ABB RobotStudio station: Braižymas_Paletavimas_V_Januška.rspag

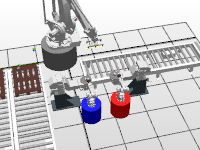
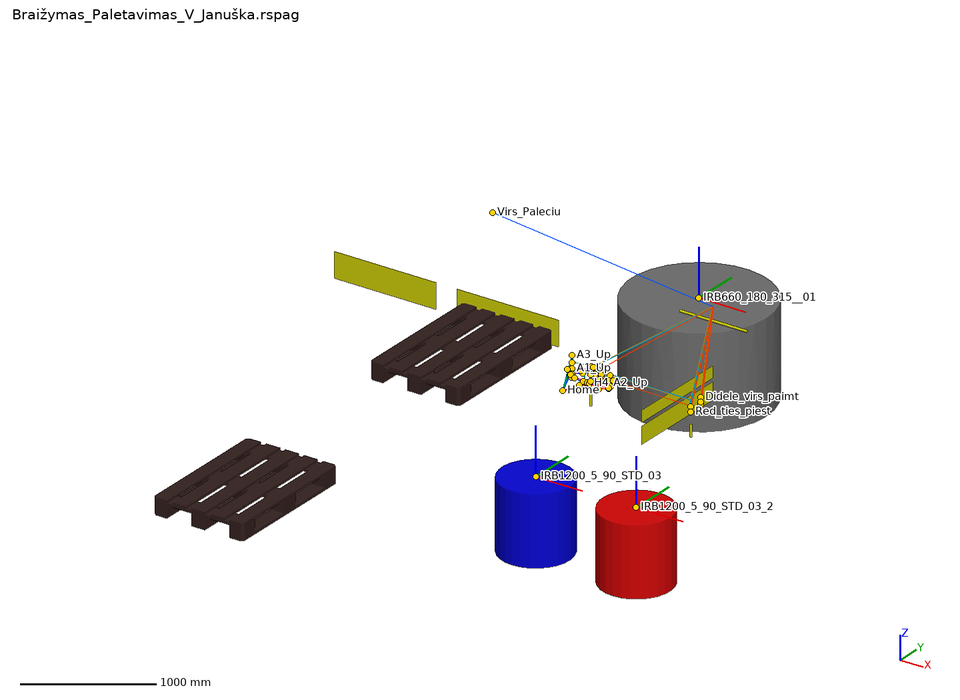
[picture v1: parts stored in the station drawn from their meshes, with robot base, taught points and paths (robot models come from the ABB library and are not in the file)]
--- station ---
Station Braižymas_Paletavimas_V_Januška (saved by RobotStudio 21.4.9700.0)
Controller Paint_Red, task T_ROB1: task frame (RAPID world) sits at (1200, -2800, 600) mm, rotated rx 0 ry 0 rz 90 deg in the station
Controller Paint_Blue, task T_ROB1: task frame (RAPID world) sits at (300, -2800, 600) mm, rotated rx 0 ry 0 rz 90 deg in the station
Controller Paletavimas, task T_ROB1: task frame (RAPID world) sits at (-200, 0, 0) mm, rotated rx 0 ry 0 rz 180 deg in the station
Controller Paletavimas
  mechanical unit ROB_1: IRB660_180_315__01, 6 joints, base frame (0, 0, 800) mm
Controller Paint_Blue
  mechanical unit ROB_1: IRB1200_5_90_STD_03, 6 joints, base frame (0, 0, 0) mm
Controller Paint_Red
  mechanical unit ROB_1: IRB1200_5_90_STD_03_2, 6 joints, base frame (0, 0, 0) mm
Layout (positions relative to the parent item):
  - IRB660_180_315__01 [mechanism] at (-200, 0, 800) mm, rotated rx 0 ry 0 rz 180 deg; joint values [2.2494, 0.0329, 0.7758, 0.6816] (rad or m)
      links: Base, Link1, Link2, Link3, LinkD1, LinkD2, LinkS1, LinkS2, Link4, LinkS3, Link6, LinkS4, LinkS5
  - Pakyla [part] at (-200, 0, 0) mm, size 1200 x 1200 x 800 mm
  - Conveyor_EUR_SC [smart component] at (-1000, -4700, 0) mm, rotated rx 0 ry 0 rz 90 deg
      signals: DI DI_New_Box, DO DO_Box_In_Place, DI DI_Delete_Pallet
      connections:
        Conveyor_EUR_SC.DI_New_Box -> PalletSource.Execute
        PalletSource.Executed -> PalletQueue.Enqueue
        PalletPlaneSensor.SensorOut -> PalletQueue.Dequeue
        PalletPlaneSensor.SensorOut -> Conveyor_EUR_SC.DO_Box_In_Place
        PalletPlaneSensor.SensorOut -> LogicGate.InputA
        LogicGate.Output -> PalletSource.Execute
        Conveyor_EUR_SC.DI_Delete_Pallet -> Sink.Execute
        PalletSource.Copy => PalletQueue.Back
        PalletPlaneSensor.SensedPart => Sink.Object
    - 950_4000_h2 [part, from Equipment\Conveyor 950 4000 h2.rslib]
    - PalletSource [smart component, from Components\Source.rslib] at (90, 55, 415) mm
        properties: Source=Euro Pallet; Copy=(none); Parent=(none); Position=[0.09 0.055 0.415]; Orientation=[0 0 0]; Transient=false; PhysicsBehavior=0
    - PalletQueue [smart component, from Components\Queue.rslib]
        properties: Back=(none); Front=(none); Queue={971251d9-3e66-4420-9243-4213e4a19f12}; NumberOfObjects=1
    - PalletPlaneSensor [smart component, from Components\PlaneSensor.rslib]
        properties: Origin=[4.05 0 0.436]; Axis1=[0 0.91 0]; Axis2=[0 0 0.22]; SensedPart=Body 1
      - _sensorPart_ [part], size 0 x 910 x 220 mm
    - LogicGate [smart component, from Components\LogicGate.rslib]
        properties: Operator=NOT; Delay=0
    - LinearMover [smart component, from Components\LinearMover.rslib]
        properties: Object=PalletQueue; Direction=[0 0.001 0]; Speed=1.2; Reference=Global; ReferenceObject=(none)
    - Euro Pallet [graphiccomponentgroup] at (90, 55, 415) mm
      - Body 1 [part], size 1200 x 800 x 144 mm
    - Sink [smart component, from Components\Sink.rslib]
        properties: Object=Body 1
    - Euro Pallet_2 [graphiccomponentgroup] at (2854.8, 55, 415) mm
      - Body 1 [part], size 1200 x 800 x 144 mm
  - Conveyor_EUR_Tall_SC [smart component] at (-2100, -4700, 0) mm, rotated rx 0 ry 0 rz 90 deg
      signals: DI DI_New_Box, DO DO_Box_In_Place, DI DI_Delete_Pallet
      connections:
        Conveyor_EUR_Tall_SC.DI_New_Box -> PalletSource.Execute
        PalletSource.Executed -> PalletQueue.Enqueue
        PalletPlaneSensor.SensorOut -> PalletQueue.Dequeue
        PalletPlaneSensor.SensorOut -> Conveyor_EUR_Tall_SC.DO_Box_In_Place
        PalletPlaneSensor.SensorOut -> LogicGate.InputA
        LogicGate.Output -> PalletSource.Execute
        Conveyor_EUR_Tall_SC.DI_Delete_Pallet -> Sink.Execute
        PalletSource.Copy => PalletQueue.Back
        PalletPlaneSensor.SensedPart => Sink.Object
    - 950_4000_h2 [part, from Equipment\Conveyor 950 4000 h2.rslib]
    - PalletSource [smart component, from Components\Source.rslib] at (90, 55, 415) mm
        properties: Source=Euro Pallet; Copy=Euro Pallet_6; Parent=(none); Position=[0.09 0.055 0.415]; Orientation=[0 0 0]; Transient=false; PhysicsBehavior=0
    - PalletQueue [smart component, from Components\Queue.rslib]
        properties: Back=Euro Pallet_6; Front=(none); Queue=; NumberOfObjects=0
    - PalletPlaneSensor [smart component, from Components\PlaneSensor.rslib]
        properties: Origin=[4.05 0 0.436]; Axis1=[0 0.91 0]; Axis2=[0 0 0.22]; SensedPart=Body 1
      - _sensorPart_ [part], size 0 x 910 x 220 mm
    - LogicGate [smart component, from Components\LogicGate.rslib]
        properties: Operator=NOT; Delay=0
    - LinearMover [smart component, from Components\LinearMover.rslib]
        properties: Object=PalletQueue; Direction=[0 0.001 0]; Speed=1.2; Reference=Global; ReferenceObject=(none)
    - Euro Pallet [graphiccomponentgroup, from Equipment\Euro Pallet.rslib] at (90, 55, 415) mm
      - Body 1 [part, from Equipment\Euro Pallet.rslib]
    - Sink [smart component, from Components\Sink.rslib]
        properties: Object=Body 1
    - Euro Pallet_6 [graphiccomponentgroup, from Equipment\Euro Pallet.rslib] at (2854.8, 55, 415) mm
      - Body 1 [part, from Equipment\Euro Pallet.rslib]
  - Pakyla_2 [part] at (300, -2800, 0) mm, rotated rx 0 ry 0 rz -90 deg, size 600 x 599 x 600 mm
  - Pakyla_3 [part] at (3000, -1800, 0) mm, rotated rx 0 ry 0 rz -90 deg, size 600 x 599 x 600 mm
  - Griebtuvas_2 [smart component] at (-790.8, -1192.17, 822.02) mm
      signals: DI DI_Attach, DI DI_Enque_Tall, DI DI_Enque_Small, DI DI_Delete_Small, DI DI_Delete_Tall
      connections:
        Griebtuvas_2.DI_Attach -> PoseMover_2.Execute
        Griebtuvas_2.DI_Attach -> Attacher.Execute
        Griebtuvas_2.DI_Attach -> LogicGate.InputA
        LogicGate.Output -> Detacher.Execute
        Griebtuvas_2.DI_Enque_Tall -> Delete_Tall_Queue.Enqueue
        Griebtuvas_2.DI_Enque_Small -> Delete_Small_Queue.Enqueue
        Griebtuvas_2.DI_Delete_Small -> Delete_Small_Queue.DeleteAll
        Griebtuvas_2.DI_Delete_Tall -> Delete_Tall_Queue.DeleteAll
        LineSensor.SensedPart => Detacher.Child
        LineSensor.SensedPart => Attacher.Child
        LineSensor.SensedPart => Delete_Small_Queue.Back
        LineSensor.SensedPart => Delete_Tall_Queue.Back
    - Attacher [smart component, from Components\Attacher.rslib] at (1573.68, -26.65, 864.9) mm, rotated rx 180 ry 0 rz 89.83 deg
        properties: Parent=Griebtuvas_2; Flange=0; Child=(none); Mount=false; Offset=[0 0 0]; Orientation=[0 0 0]
    - Detacher [smart component, from Components\Detacher.rslib] at (1573.68, -26.65, 864.9) mm, rotated rx 180 ry 0 rz 89.83 deg
        properties: Child=(none); KeepPosition=true
    - LineSensor [smart component, from Components\LineSensor.rslib] at (1573.68, -26.65, 864.9) mm, rotated rx 180 ry 0 rz 89.83 deg
        properties: Start=[-6.04715178049997E-07 0.300000227208211 0.311447110706865]; End=[-3.13979206786885E-07 -0.300000333635623 0.311447110706865]; Radius=0.01; SensedPart=(none); SensedPoint=[0 0 0]
      - _sensorPart_ [part], size 20 x 600 x 20 mm
    - VacuumTool [mechanism] at (1573.68, -26.65, 864.9) mm, rotated rx 180 ry 0 rz 89.83 deg
        TCP tVacuum at (0, 0, 200) mm
        links: VacuumTool
    - LogicGate [smart component, from Components\LogicGate.rslib]
        properties: Operator=NOT; Delay=0
    - Delete_Small_Queue [smart component, from Components\Queue.rslib]
        properties: Back=(none); Front=(none); Queue=; NumberOfObjects=0
    - Delete_Tall_Queue [smart component, from Components\Queue.rslib]
        properties: Back=(none); Front=(none); Queue=; NumberOfObjects=0
  - Pozicionierius_Red [smart component] at (1200, -2100, 0) mm
      signals: DI DI_Attach, DO DO_Attached, DI DI_TurnR, DI DI_TurnL, DO DO_Complete, DI DI_Home, DO DO_Free
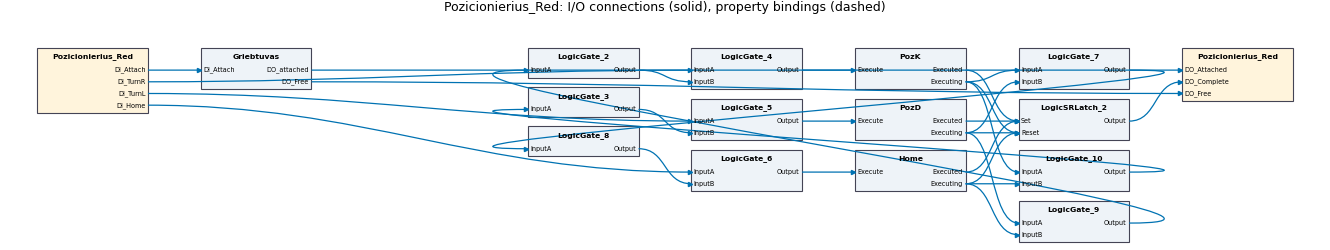
      connections:
        Pozicionierius_Red.DI_Attach -> Griebtuvas.DI_Attach
        Griebtuvas.DO_attached -> Pozicionierius_Red.DO_Attached
        LogicGate_4.Output -> PozK.Execute
        LogicGate_5.Output -> PozD.Execute
        LogicGate_6.Output -> Home.Execute
        Pozicionierius_Red.DI_TurnR -> LogicGate_4.InputA
        Pozicionierius_Red.DI_TurnL -> LogicGate_5.InputA
        Pozicionierius_Red.DI_Home -> LogicGate_6.InputA
        LogicSRLatch_2.Output -> Pozicionierius_Red.DO_Complete
        PozK.Executed -> LogicSRLatch_2.Set
        PozD.Executed -> LogicSRLatch_2.Set
        Home.Executed -> LogicSRLatch_2.Set
        PozK.Executing -> LogicGate_7.InputA
        PozK.Executing -> LogicGate_10.InputA
        PozD.Executing -> LogicGate_7.InputB
        PozD.Executing -> LogicGate_9.InputA
        Home.Executing -> LogicGate_9.InputB
        Home.Executing -> LogicGate_10.InputB
        LogicGate_9.Output -> LogicGate_2.InputA
        LogicGate_10.Output -> LogicGate_3.InputA
        LogicGate_7.Output -> LogicGate_8.InputA
        LogicGate_2.Output -> LogicGate_4.InputB
        LogicGate_3.Output -> LogicGate_5.InputB
        LogicGate_8.Output -> LogicGate_6.InputB
        Home.Executing -> LogicSRLatch_2.Reset
        PozD.Executing -> LogicSRLatch_2.Reset
        PozK.Executing -> LogicSRLatch_2.Reset
        Griebtuvas.DO_Free -> Pozicionierius_Red.DO_Free
    - Griebtuvas [smart component]
        signals: DI DI_Attach, DO DO_attached, DO DO_Free
        connections:
          Griebtuvas.DI_Attach -> Attacher.Execute
          Griebtuvas.DI_Attach -> LogicGate.InputA
          LogicGate.Output -> Detacher.Execute
          Attacher.Executed -> LogicSRLatch.Set
          Detacher.Executed -> LogicSRLatch.Reset
          LogicSRLatch.Output -> Griebtuvas.DO_attached
          LineSensor.SensorOut -> LogicGate_2.InputA
          LogicGate_2.Output -> Griebtuvas.DO_Free
          LineSensor.SensedPart => Attacher.Child
          LineSensor.SensedPart => Detacher.Child
      - Attacher [smart component, from Components\Attacher.rslib]
          properties: Parent=IRBP_A250_D1000_M2009_REV1_01; Flange=0; Child=(none); Mount=false; Offset=[0 0 0]; Orientation=[0 0 0]
      - Detacher [smart component, from Components\Detacher.rslib]
          properties: Child=(none); KeepPosition=true
      - LogicGate [smart component, from Components\LogicGate.rslib]
          properties: Operator=NOT; Delay=0
      - LogicSRLatch [smart component, from Components\LogicSRLatch.rslib]
      - LineSensor [smart component, from Components\LineSensor.rslib]
          properties: Start=[0 0 0.9]; End=[0 0 1]; Radius=0.01; SensedPart=(none); SensedPoint=[0 0 0]
        - _sensorPart_ [part], size 20 x 20 x 100 mm
      - LogicGate_2 [smart component, from Components\LogicGate.rslib]
          properties: Operator=NOT; Delay=0
    - IRBP_A250_D1000_M2009_REV1_01 [mechanism] at (0, 0, 0) mm; joint values [0, 1.5708] (rad or m)
        links: Base, Link1, Link2
    - PozD [smart component, from Components\PoseMover.rslib]
        properties: Mechanism=IRBP_A250_D1000_M2009_REV1_01; Pose=2; Duration=0.5
    - PozK [smart component, from Components\PoseMover.rslib]
        properties: Mechanism=IRBP_A250_D1000_M2009_REV1_01; Pose=3; Duration=0.5
    - Home [smart component, from Components\PoseMover.rslib]
        properties: Mechanism=IRBP_A250_D1000_M2009_REV1_01; Pose=1; Duration=0.5
    - LogicGate_2 [smart component, from Components\LogicGate.rslib]
        properties: Operator=NOT; Delay=0
    - LogicGate_3 [smart component, from Components\LogicGate.rslib]
        properties: Operator=NOT; Delay=0
    - LogicGate_4 [smart component, from Components\LogicGate.rslib]
        properties: Operator=AND; Delay=0
    - LogicGate_5 [smart component, from Components\LogicGate.rslib]
        properties: Operator=AND; Delay=0
    - LogicGate_6 [smart component, from Components\LogicGate.rslib]
        properties: Operator=AND; Delay=0
    - LogicGate_7 [smart component, from Components\LogicGate.rslib]
        properties: Operator=OR; Delay=0
    - LogicGate_8 [smart component, from Components\LogicGate.rslib]
        properties: Operator=NOT; Delay=0
    - LogicGate_9 [smart component, from Components\LogicGate.rslib]
        properties: Operator=OR; Delay=0
    - LogicGate_10 [smart component, from Components\LogicGate.rslib]
        properties: Operator=OR; Delay=0
    - LogicSRLatch_2 [smart component, from Components\LogicSRLatch.rslib]
  - Pozicionierius_Blue [smart component] at (300, -2100, 0) mm, rotated rx 0 ry 0 rz 180 deg
      signals: DI DI_Attach, DO DO_Attached, DI DI_TurnR, DI DI_TurnL, DO DO_Complete, DI DI_Home, DO DO_Free
      connections:
        Pozicionierius_Blue.DI_Attach -> Griebtuvas.DI_Attach
        Griebtuvas.DO_attached -> Pozicionierius_Blue.DO_Attached
        LogicGate_4.Output -> PozK.Execute
        LogicGate_5.Output -> PozD.Execute
        LogicGate_6.Output -> Home.Execute
        Pozicionierius_Blue.DI_TurnR -> LogicGate_4.InputA
        Pozicionierius_Blue.DI_TurnL -> LogicGate_5.InputA
        Pozicionierius_Blue.DI_Home -> LogicGate_6.InputA
        LogicSRLatch_2.Output -> Pozicionierius_Blue.DO_Complete
        PozK.Executed -> LogicSRLatch_2.Set
        PozD.Executed -> LogicSRLatch_2.Set
        Home.Executed -> LogicSRLatch_2.Set
        PozK.Executing -> LogicGate_7.InputA
        PozK.Executing -> LogicGate_10.InputA
        PozD.Executing -> LogicGate_7.InputB
        PozD.Executing -> LogicGate_9.InputA
        Home.Executing -> LogicGate_9.InputB
        Home.Executing -> LogicGate_10.InputB
        LogicGate_9.Output -> LogicGate_2.InputA
        LogicGate_10.Output -> LogicGate_3.InputA
        LogicGate_7.Output -> LogicGate_8.InputA
        LogicGate_2.Output -> LogicGate_4.InputB
        LogicGate_3.Output -> LogicGate_5.InputB
        LogicGate_8.Output -> LogicGate_6.InputB
        Home.Executing -> LogicSRLatch_2.Reset
        PozD.Executing -> LogicSRLatch_2.Reset
        PozK.Executing -> LogicSRLatch_2.Reset
        Griebtuvas.DO_Free -> Pozicionierius_Blue.DO_Free
    - Griebtuvas [smart component]
        signals: DI DI_Attach, DO DO_attached, DO DO_Free
        connections:
          Griebtuvas.DI_Attach -> Attacher.Execute
          Griebtuvas.DI_Attach -> LogicGate.InputA
          LogicGate.Output -> Detacher.Execute
          Attacher.Executed -> LogicSRLatch.Set
          Detacher.Executed -> LogicSRLatch.Reset
          LogicSRLatch.Output -> Griebtuvas.DO_attached
          LineSensor.SensorOut -> LogicGate_3.InputA
          LogicGate_3.Output -> Griebtuvas.DO_Free
          LineSensor.SensedPart => Attacher.Child
          LineSensor.SensedPart => Detacher.Child
          LineSensor.SensedPart => Detacher.Child
          LineSensor.SensedPart => Attacher.Child
      - Attacher [smart component, from Components\Attacher.rslib]
          properties: Parent=IRBP_A250_D1000_M2009_REV1_01; Flange=0; Child=(none); Mount=false; Offset=[0 0 0]; Orientation=[0 0 0]
      - Detacher [smart component, from Components\Detacher.rslib]
          properties: Child=(none); KeepPosition=true
      - LogicGate [smart component, from Components\LogicGate.rslib]
          properties: Operator=NOT; Delay=0
      - LogicSRLatch [smart component, from Components\LogicSRLatch.rslib]
      - LineSensor [smart component, from Components\LineSensor.rslib]
          properties: Start=[0 0 0.9]; End=[0 0 1]; Radius=0.01; SensedPart=(none); SensedPoint=[0 0 0]
        - _sensorPart_ [part], size 20 x 20 x 100 mm
      - LogicGate_3 [smart component, from Components\LogicGate.rslib]
          properties: Operator=NOT; Delay=0
    - IRBP_A250_D1000_M2009_REV1_01 [mechanism] at (0, 0, 0) mm; joint values [0, 1.5708] (rad or m)
        links: Base, Link1, Link2
    - PozD [smart component, from Components\PoseMover.rslib]
        properties: Mechanism=IRBP_A250_D1000_M2009_REV1_01; Pose=2; Duration=0.5
    - PozK [smart component, from Components\PoseMover.rslib]
        properties: Mechanism=IRBP_A250_D1000_M2009_REV1_01; Pose=3; Duration=0.5
    - Home [smart component, from Components\PoseMover.rslib]
        properties: Mechanism=IRBP_A250_D1000_M2009_REV1_01; Pose=1; Duration=0.5
    - LogicGate_2 [smart component, from Components\LogicGate.rslib]
        properties: Operator=NOT; Delay=0
    - LogicGate_3 [smart component, from Components\LogicGate.rslib]
        properties: Operator=NOT; Delay=0
    - LogicGate_4 [smart component, from Components\LogicGate.rslib]
        properties: Operator=AND; Delay=0
    - LogicGate_5 [smart component, from Components\LogicGate.rslib]
        properties: Operator=AND; Delay=0
    - LogicGate_6 [smart component, from Components\LogicGate.rslib]
        properties: Operator=AND; Delay=0
    - LogicGate_7 [smart component, from Components\LogicGate.rslib]
        properties: Operator=OR; Delay=0
    - LogicGate_8 [smart component, from Components\LogicGate.rslib]
        properties: Operator=NOT; Delay=0
    - LogicGate_9 [smart component, from Components\LogicGate.rslib]
        properties: Operator=OR; Delay=0
    - LogicGate_10 [smart component, from Components\LogicGate.rslib]
        properties: Operator=OR; Delay=0
    - LogicSRLatch_2 [smart component, from Components\LogicSRLatch.rslib]
  - IRB1200_5_90_STD_03 [mechanism, from Robots\IRB1200_5_90_STD_03.rslib] at (300, -2800, 600) mm, rotated rx 0 ry 0 rz 90 deg; joint values [-0.0192, -0.8245, 0.9777, -0.1248, -0.1544, 0.1234] (rad or m)
  - IRB1200_5_90_STD_03_2 [mechanism, from Robots\IRB1200_5_90_STD_03.rslib] at (1200, -2800, 600) mm, rotated rx 0 ry 0 rz 90 deg; joint values [-0.0192, -0.8245, 0.9777, -0.1248, -0.1544, 0.1234] (rad or m)
  - Conveyor_RND_SC [smart component] at (4500, -750, 0) mm, rotated rx 0 ry 0 rz 180 deg
      signals: DI DI_New_Box, DO DO_Box_InPlace, DO DO_TallBox_InPlace, DO DO_Only_High_Sensor
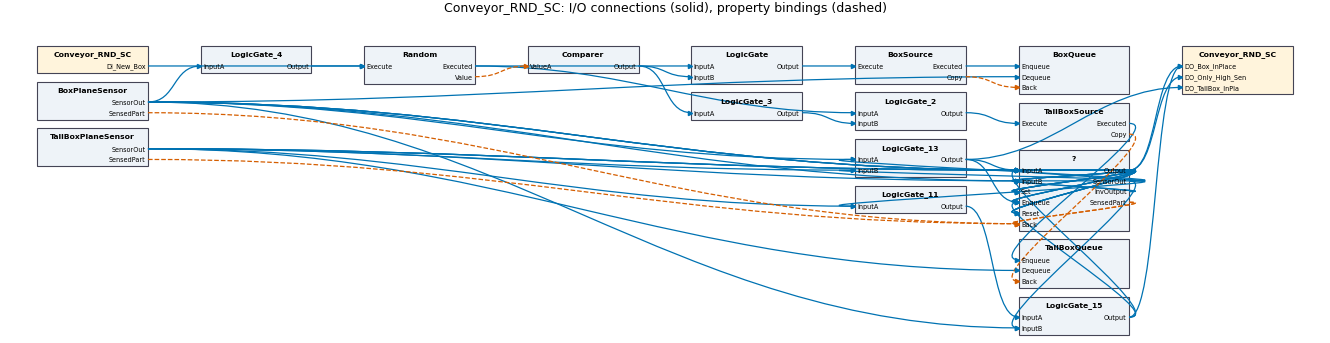
      connections:
        Conveyor_RND_SC.DI_New_Box -> Random.Execute
        Random.Executed -> LogicGate.InputA
        Random.Executed -> LogicGate_2.InputA
        Comparer.Output -> LogicGate_3.InputA
        LogicGate_3.Output -> LogicGate_2.InputB
        Comparer.Output -> LogicGate.InputB
        LogicGate.Output -> BoxSource.Execute
        LogicGate_2.Output -> TallBoxSource.Execute
        BoxSource.Executed -> BoxQueue.Enqueue
        LogicGate_4.Output -> Random.Execute
        BoxPlaneSensor.SensorOut -> LogicGate_4.InputA
        BoxPlaneSensor.SensorOut -> BoxQueue.Dequeue
        TallBoxSource.Executed -> TallBoxQueue.Enqueue
        TallBoxPlaneSensor.SensorOut -> TallBoxQueue.Dequeue
        TallBoxPlaneSensor.SensorOut -> ?.InputA
        BoxPlaneSensor.SensorOut -> ?.InputA
        ?.Output -> ?.InputB
        TallBoxPlaneSensor.SensorOut -> ?.InputA
        BoxPlaneSensor.SensorOut -> ?.InputB
        ?.Output -> ?.InputA
        ?.Output -> ?.Set
        ?.Output -> Conveyor_RND_SC.DO_Box_InPlace
        ?.Output -> Delete_Small_Queue.Enqueue
        ?.Output -> ?.Set
        ?.Output -> ?.InputA
        ?.Output -> ?.Reset
        ?.Output -> ?.InputA
        ?.Output -> ?.Reset
        ?.SensorOut -> LogicGate_13.InputA
        ?.SensorOut -> LogicGate_13.InputB
        ?.SensorOut -> LogicGate_11.InputA
        LogicGate_11.Output -> LogicGate_15.InputA
        ?.SensorOut -> LogicGate_15.InputB
        LogicGate_13.Output -> LogicGate_16.InputA
        LogicGate_16.Output -> LogicSRLatch_4.Set
        LogicGate_15.Output -> LogicGate_14.InputA
        LogicGate_14.Output -> LogicSRLatch_5.Set
        LogicSRLatch_5.InvOutput -> LogicGate_16.InputB
        LogicSRLatch_4.InvOutput -> LogicGate_14.InputB
        ?.SensorOut -> LogicGate_18.InputA
        ?.SensorOut -> LogicGate_18.InputB
        LogicGate_18.Output -> LogicGate_17.InputA
        LogicGate_17.Output -> LogicSRLatch_4.Reset
        TallBoxPlaneSensor.SensorOut -> LogicGate_18.InputB
        TallBoxPlaneSensor.SensorOut -> LogicGate_13.InputB
        TallBoxPlaneSensor.SensorOut -> LogicGate_11.InputA
        BoxPlaneSensor.SensorOut -> LogicGate_18.InputA
        BoxPlaneSensor.SensorOut -> LogicGate_13.InputA
        BoxPlaneSensor.SensorOut -> LogicGate_15.InputB
        LogicSRLatch_5.Output -> LogicGate_19.InputB
        LogicGate_19.Output -> Delete_Small_Queue.Enqueue
        LogicGate_20.Output -> Delete_Tall_Queue.Enqueue
        LogicSRLatch_4.Output -> LogicGate_20.InputB
        LogicGate_23.Output -> LogicGate_21.InputB
        BoxPlaneSensor.SensorOut -> LogicGate_23.InputA
        TallBoxPlaneSensor.SensorOut -> LogicGate_21.InputA
        LogicGate_21.Output -> LogicGate_19.InputA
        LogicGate_21.Output -> LogicGate_20.InputA
        LogicGate_21.Output -> Conveyor_RND_SC.DO_Only_High_Sensor
        LogicGate_17.Output -> LogicSRLatch_5.Reset
        LogicGate_13.Output -> Conveyor_RND_SC.DO_TallBox_InPlace
        LogicGate_15.Output -> Conveyor_RND_SC.DO_Box_InPlace
        LogicGate_15.Output -> Delete_Small_Queue.Enqueue
        LogicGate_13.Output -> Delete_Tall_Queue.Enqueue
        Random.Value => Comparer.ValueA
        BoxSource.Copy => BoxQueue.Back
        TallBoxSource.Copy => TallBoxQueue.Back
        DeleteSensor.SensedPart => Delete_Small_Queue.Back
        DeleteSensor.SensedPart => Delete_Tall_Queue.Back
        BoxPlaneSensor.SensedPart => Delete_Small_Queue.Back
        TallBoxPlaneSensor.SensedPart => Delete_Tall_Queue.Back
    - 950_4000 [part, from Equipment\Conveyor 950 4000 h2.rslib]
    - Box [part] at (60, 300, 415) mm, size 500 x 300 x 200 mm
    - BoxPlaneSensor [smart component, from Components\PlaneSensor.rslib]
        properties: Origin=[4.05 0 0.45]; Axis1=[0 0.91 0]; Axis2=[0 0 0.15]; SensedPart=(none)
      - _sensorPart_ [part], size 0 x 910 x 150 mm
    - BoxQueue [smart component, from Components\Queue.rslib] at (0, -3000, 0) mm
        properties: Back=(none); Front=(none); Queue={fa6990f4-df59-49ae-9a32-9599613f68ec};{e767133d-be7e-453b-8722-821a6b4558c0};{6ce431a7-dd26-4a38-b4fa-eec74b1977cf};{3ae16747-654e-4202-adcd-dee3cf7f9746};{658dea4e-2eb4-4657-ae88-8a3f4d155435};{5f69d4f6-3337-4fea-9838-df10eb0f07de};{5aecbc6f-cfd0-44df-ba1d-f4507ba342ea};{9e44f664-69de-4a1f-8895-3168aa3968ee};{5f2001e6-6928-42db-81b0-89c8c28d3b67};{af1fb1b9-f86a-429e-8c15-d7efb4d2c7e7};{8385d1b0-8c34-4fb9-9887-15fbe6147db4};{4006f633-1bd4-4d72-a937-3620dfa0b835};{8730c694-ac09-41e2-b981-cff9bcc11746};{a723061a-c6e3-4254-9954-9e38f42a9860};{04c40ebc-cfd0-4884-a185-3f6b111fdaa2};{a878a6d6-609e-42c1-80c8-878f67ab97da};{14d7b2c0-999e-4cbf-889d-0a124069ec19};{0becc2c0-5e92-4cfa-b639-036a75e5a4e4};{cca5aef1-b22d-4971-98ab-11323a0a7094};{e02a7358-ec92-4485-b2c0-c2038150d912};{6839aee3-4009-4411-9cbe-94a25d9f948c};{9f3facf0-270c-4be3-a67a-821ea0c5aa08};{faba08c9-aeb2-4eb9-b9c7-e387a6e9cbfb};{bc03e252-87de-4255-9640-78523ef2143d};{aa76d2e2-ad85-4407-8279-2d879163961a};{be818020-9745-4898-a081-c1837189eb10};{37e33ad3-8b58-4812-a8ee-bee1f17e24b7};{41a75c38-fc95-4d9b-aee3-f79fb853da63};{f3c5d293-df41-45c9-8c8c-c5c112b7c860};{0c1f799b-0fa7-450f-a03e-204d5134bc88};{4de367fb-fa00-4147-a461-8cdc53a5ab36};{fb4f46fb-3cc9-46d0-93b3-3697bff4c5b0};{1981477c-fa3d-405d-81ed-5c11cf4004f1};{4a3acb3a-f0fe-49f4-bb5a-d33d1ebb5bdb};{ee543a3a-f0a7-4b8a-ba73-df8df06667eb};{37d46d93-7b88-48c0-95e4-0c0aea62eed6};{e38b9446-edb0-4063-af88-28e337124caa};{43dc83e6-1610-4f95-90e3-0b23558226fe};{ea22c4f6-820c-436e-a9cf-17bec50e4e45};{7837ae08-a857-4e45-b104-d71f85b8db14};{a15a4319-5ddc-4b41-a9f1-f3fc310fac6a};{fcbb5e9a-b5e8-401e-bfdc-b057d8770794};{ce142922-48a3-4377-89ec-985408ba8153};{9c2054a3-2d81-4b78-8319-3879110db110};{4184086f-4b9b-435c-872e-61dbf8e8b281};{2e9da51f-8d60-4fa4-b223-03c706fc42b4};{f081e902-d69f-44bb-8e7e-e42cb8ba28a7};{0c45a0ca-c831-4e04-b0c0-ea9f274c986f};{68cd1851-b56a-466d-8aa0-fcc04310c142};{8d21e733-4511-40ca-a380-e002fb2e741f};{1fdcc6e5-ab2a-4a16-b63c-6443d12e6cd0};{928b3c83-786f-4b1b-b774-b6e363eb8edd};{c5d4ec7b-f50e-4586-9c9a-3cfc5369afde};{176768ad-9249-4043-a0f4-b263c87cbf02};{a41bf4c8-ca06-40df-8d99-855080af08cc};{1f7c0284-63bf-491f-a88a-99226beab572};{93b63075-c389-479b-b9ba-db424c8f1608};{46184e33-de41-46df-bfa5-1fa5c4186c93};{ff1b25a2-d9f1-4991-8a41-ba89a23b8150};{72555af7-e6df-461e-9b88-b16b7a0d81b3};{b15f7b76-8d34-4692-97fc-69f520f0f3c0};{93a6a054-f8ca-4001-a03b-5df487de4b8b};{72ed48d2-5bfa-4ecc-a1ec-2e7778b8ef55};{9cda9d10-0121-4b20-9212-f063ab80550a};{33ea0952-9bf3-4e06-b34c-2e0ac0a36824};{e1a11204-25f8-485f-a139-3d4a140b070a};{3c953577-cf61-4183-9ff0-bca456af431b};{30fbd990-83ea-4ba2-9465-f98aa0538540};{dfe653b7-7d94-4ddd-b2ef-7199ad70201c};{82d208d8-4dee-4044-8917-702fcaee31aa};{aa19c751-7ff3-4b4e-bfb3-31ee09fcbfd8};{cfec794f-833e-41bb-b0d0-1a3d28b30ff6};{6a23a3bd-1c81-490c-bc0d-d6dcbd6c3643};{8a1ebaad-f4c7-4178-a576-8aee444642b5};{ba785cc5-e159-446c-93f0-7483d17038e5};{828e2240-582c-4548-b989-1a7bc8d860a3};{4a59a418-7f0b-41e9-93ce-595c45a59b07};{f4dbaa99-1c72-4e73-8856-0fc6635ef423};{6087b47d-53c7-4741-b2a3-0c083e370b15};{2e30bba9-a6bf-4b01-9fc0-a1f4cbfc7dfc};{19071a2c-5ad0-42a1-9bd2-bb839ae9b4d4};{b0002f64-93e0-428c-b2e5-2d4d9f7da933};{a347c7fd-09d1-4374-ab85-2149f88733a9};{b0d38dbd-07a6-4783-b2e8-5f2c5d6b0201};{2266d51d-b3d0-4d52-bbb5-de615e632cc2};{75460951-9708-49ff-8c70-7d7735d8d5c2};{295ff81f-2104-47a7-8bd3-4eaad3dc957a};{0a807d55-7f1b-46ac-9050-abab5979a08e};{896dd1f3-c715-442d-b525-9d9e6cb6e06f};{4fa8727e-168a-49f4-b20a-f869ddebea6d};{9c068a76-23d8-4921-84fc-952de2f64cfe};{4b6f13b1-b58b-4cfc-9d2f-06395fabde15};{01d6ab25-4f5e-4e9f-bdfc-4dfebc0f0cf6};{0ab7461e-d2ad-4383-836c-68a8b79c7dca};{06b8ba49-82c0-4634-8553-9497b791d1b9};{f3c0ef50-404a-451a-a529-2526a8561f87};{0ffca263-bbd3-4c7e-912c-55349d3e2daa};{252a513a-a084-4872-865a-129838c2f94f};{466e5942-a908-47e1-8cd1-136cfa812536};{1b8b29c7-edcf-413e-9f81-164808a08126};{5c9bba4a-b90c-47ae-95ca-d31383bcbc95};{a37f6f99-c3a3-4e91-9e81-52d69c79e6c0};{eaa8d07c-22f4-4512-a4ed-d3e2fd25e17b};{cd5a02a4-7d6b-4818-9494-1cca1ee745c5};{c0bf9634-2c95-4f7a-b6ff-e31064599eb0};{8cba37ce-13ba-401a-b10d-a55bd7da9434};{350e1ddc-e127-4834-bdb0-6da9a5ae8f39};{12ff0c17-9d1a-4539-a0c4-b273c13be77a};{36d11481-6af8-4316-a391-be7944f9a913};{9e99407b-b875-4dbb-ac3e-7ed2c2198c50};{18fd7586-1f58-49bb-aa86-4785e5672a8a};{4590a0b8-4fa4-4fd5-96ec-6588471226b3};{0910f9d0-3289-4e14-ada6-3d436962069f};{6e596c34-5dbf-4a37-9b92-6d9d57f91504};{2fc5be82-8ebc-4497-b7a2-a92180d8126c};{e572f00d-1eb5-4a34-a751-0ba51d1a1975};{68969745-703d-4f84-abfd-8cca6df6441f};{bd9b3794-10fd-4df4-8bef-e9c82c14e8cf};{f3ae70ba-db38-470f-8edb-540b6fe1d8be};{2a3c6a5a-be7f-42bd-82e9-81bfd16108a1};{25c3ed99-c921-4982-a94c-124f118646ae}; NumberOfObjects=1
    - BoxSource [smart component, from Components\Source.rslib] at (0, -3000, 0) mm
        properties: Source=Box; Copy=(none); Parent=(none); Position=[0.06 0.325 0.415]; Orientation=[0 0 0]; Transient=false; PhysicsBehavior=0
    - LinearMover [smart component, from Components\LinearMover.rslib] at (0, -3000, 0) mm
        properties: Object=BoxQueue; Direction=[-0.001 0 0]; Speed=1.2; Reference=Global; ReferenceObject=(none)
    - Random [smart component, from Components\Random.rslib] at (3800, -500, 0) mm, rotated rx 0 ry 0 rz 180 deg
        properties: Value=0.429773476640588; Min=0; Max=1
    - Comparer [smart component, from Components\Comparer.rslib] at (3800, -500, 0) mm, rotated rx 0 ry 0 rz 180 deg
        properties: ValueA=0.429773476640588; Operator=>=; ValueB=0.5
    - TallBoxSource [smart component, from Components\Source.rslib] at (0, -3000, 0) mm
        properties: Source=Box_tall; Copy=(none); Parent=(none); Position=[0.06 0.325 0.415]; Orientation=[0 0 0]; Transient=false; PhysicsBehavior=0
    - LogicGate [smart component, from Components\LogicGate.rslib] at (3800, -500, 0) mm, rotated rx 0 ry 0 rz 180 deg
        properties: Operator=AND; Delay=0
    - LogicGate_2 [smart component, from Components\LogicGate.rslib] at (3800, -500, 0) mm, rotated rx 0 ry 0 rz 180 deg
        properties: Operator=AND; Delay=0
    - LogicGate_3 [smart component, from Components\LogicGate.rslib] at (3800, -500, 0) mm, rotated rx 0 ry 0 rz 180 deg
        properties: Operator=NOT; Delay=0
    - LogicGate_4 [smart component, from Components\LogicGate.rslib] at (3800, -500, 0) mm, rotated rx 0 ry 0 rz 180 deg
        properties: Operator=NOT; Delay=0
    - TallBoxPlaneSensor [smart component, from Components\PlaneSensor.rslib]
        properties: Origin=[4.05 0 0.63]; Axis1=[0 0.91 0]; Axis2=[0 0 0.1]; SensedPart=(none)
      - _sensorPart_ [part], size 0 x 910 x 100 mm
    - Box_tall [part] at (60, 300, 415) mm, size 500 x 300 x 250 mm
    - TallBoxQueue [smart component, from Components\Queue.rslib]
        properties: Back=(none); Front=(none); Queue=; NumberOfObjects=0
    - LinearMover_2 [smart component, from Components\LinearMover.rslib]
        properties: Object=TallBoxQueue; Direction=[-0.001 0 0]; Speed=1.2; Reference=Global; ReferenceObject=(none)
    - LogicGate_10 [smart component, from Components\LogicGate.rslib]
        properties: Operator=AND; Delay=0
    - LogicGate_11 [smart component, from Components\LogicGate.rslib]
        properties: Operator=NOT; Delay=0
    - LogicGate_12 [smart component, from Components\LogicGate.rslib]
        properties: Operator=AND; Delay=0
    - LogicGate_13 [smart component, from Components\LogicGate.rslib]
        properties: Operator=AND; Delay=0
    - LogicGate_15 [smart component, from Components\LogicGate.rslib]
        properties: Operator=AND; Delay=0
  - TraceTCP [smart component, from Components\TraceTCP.rslib]
      properties: Robot=IRB1200_5_90_STD_03
  - TraceTCP_2 [smart component, from Components\TraceTCP.rslib]
      properties: Robot=IRB1200_5_90_STD_03_2
  - Pen_Blue [mechanism, from Training Objects\Pen.rslib] at (302.36, -2594.82, 1275.93) mm, rotated rx 0 ry 90 rz 90 deg
  - Pen_Red [mechanism, from Training Objects\Pen.rslib] at (1202.36, -2594.82, 1275.93) mm, rotated rx 0 ry 90 rz 90 deg
Attachment: VacuumTool is attached to IRB660_180_315__01 / Link6
Attachment: Griebtuvas_2 is attached to IRB660_180_315__01 / Link6
Attachment: TallBoxSource is attached to BoxSource
Attachment: Pen_Blue is attached to IRB1200_5_90_STD_03 / Link6
Attachment: Pen_Red is attached to IRB1200_5_90_STD_03_2 / Link6
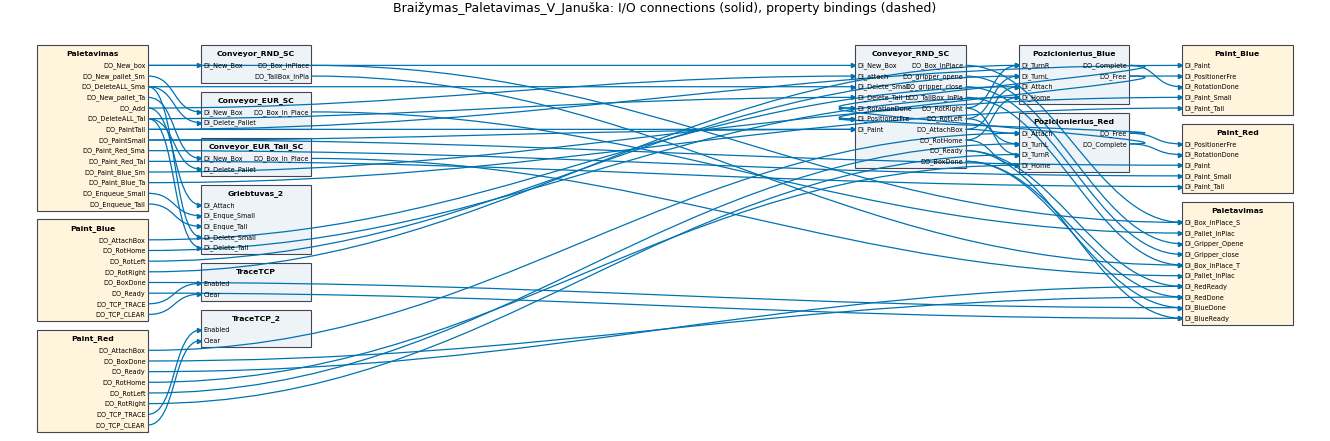
Station logic (signal -> signal, property => property):
  Paletavimas.DO_New_box -> Conveyor_RND_SC.DI_New_Box
  Paletavimas.DO_New_pallet_Small -> Conveyor_EUR_SC.DI_New_Box
  Conveyor_RND_SC.DO_Box_InPlace -> Paletavimas.DI_Box_InPlace_Small
  Conveyor_EUR_SC.DO_Box_In_Place -> Paletavimas.DI_Pallet_InPlace_Small
  Griebtuvas_SC.DO_gripper_opened -> Paletavimas.DI_Gripper_Opened
  Griebtuvas_SC.DO_gripper_closed -> Paletavimas.DI_Gripper_closed
  Paletavimas.DO_DeleteALL_Small -> Conveyor_EUR_SC.DI_Delete_Pallet
  Paletavimas.DO_New_pallet_Tall -> Conveyor_EUR_Tall_SC.DI_New_Box
  Conveyor_RND_SC.DO_TallBox_InPlace -> Paletavimas.DI_Box_InPlace_Tall
  Conveyor_EUR_Tall_SC.DO_Box_In_Place -> Paletavimas.DI_Pallet_InPlace_Tall
  Paletavimas.DO_Add -> Griebtuvas_SC.DI_attach
  Paletavimas.DO_DeleteALL_Tall -> Conveyor_EUR_Tall_SC.DI_Delete_Pallet
  Paletavimas.DO_DeleteALL_Small -> Conveyor_RND_SC.DI_Delete_Small_boxes
  Paletavimas.DO_DeleteALL_Tall -> Conveyor_RND_SC.DI_Delete_Tall_boxes
  Piesimas_Blue.DO_RotRight -> Pozicionierius_Blue.DI_TurnR
  Piesimas_Blue.DO_RotLeft -> Pozicionierius_Blue.DI_TurnL
  Piesimas_Red.DO_AttachBox -> Pozicionierius_Red.DI_Attach
  Piesimas_Blue.DO_AttachBox -> Pozicionierius_Blue.DI_Attach
  Paletavimas.DO_Add -> Griebtuvas_2.DI_Attach
  Piesimas_Blue.DO_RotHome -> Pozicionierius_Blue.DI_Home
  Pozicionierius_Blue.DO_Complete -> Piesimas_Blue.DI_RotationDone
  Pozicionierius_Blue.DO_Free -> Piesimas_Blue.DI_PositionerFree
  Piesimas_Red.DO_RotLeft -> Pozicionierius_Red.DI_TurnL
  Piesimas_Red.DO_RotRight -> Pozicionierius_Red.DI_TurnR
  Piesimas_Red.DO_RotHome -> Pozicionierius_Red.DI_Home
  Pozicionierius_Red.DO_Free -> Piesimas_Red.DI_PositionerFree
  Pozicionierius_Red.DO_Complete -> Piesimas_Red.DI_RotationDone
  Piesimas_Red.DO_Ready -> Paletavimas.DI_RedReady
  Piesimas_Red.DO_BoxDone -> Paletavimas.DI_RedDone
  Piesimas_Blue.DO_BoxDone -> Paletavimas.DI_BlueDone
  Piesimas_Blue.DO_Ready -> Paletavimas.DI_BlueReady
  Paletavimas.DO_PaintTall -> Piesimas_Blue.DI_Paint
  Paletavimas.DO_PaintSmall -> Piesimas_Red.DI_Paint
  Paint_Blue.DO_AttachBox -> Pozicionierius_Blue.DI_Attach
  Paint_Blue.DO_RotHome -> Pozicionierius_Blue.DI_Home
  Paint_Blue.DO_RotLeft -> Pozicionierius_Blue.DI_TurnL
  Paint_Blue.DO_RotRight -> Pozicionierius_Blue.DI_TurnR
  Paint_Blue.DO_BoxDone -> Paletavimas.DI_BlueDone
  Paletavimas.DO_PaintTall -> Paint_Blue.DI_Paint
  Pozicionierius_Blue.DO_Free -> Paint_Blue.DI_PositionerFree
  Pozicionierius_Blue.DO_Complete -> Paint_Blue.DI_RotationDone
  Paint_Red.DO_AttachBox -> Pozicionierius_Red.DI_Attach
  Paint_Red.DO_BoxDone -> Paletavimas.DI_RedDone
  Paint_Red.DO_Ready -> Paletavimas.DI_RedReady
  Paint_Red.DO_RotHome -> Pozicionierius_Red.DI_Home
  Paint_Red.DO_RotLeft -> Pozicionierius_Red.DI_TurnL
  Paint_Red.DO_RotRight -> Pozicionierius_Red.DI_TurnR
  Pozicionierius_Red.DO_Free -> Paint_Red.DI_PositionerFree
  Pozicionierius_Red.DO_Complete -> Paint_Red.DI_RotationDone
  Paletavimas.DO_PaintSmall -> Paint_Red.DI_Paint
  Conveyor_RND_SC.DO_Box_InPlace -> Paletavimas.DI_Box_InPlace_Small
  Conveyor_RND_SC.DO_TallBox_InPlace -> Paletavimas.DI_Box_InPlace_Tall
  Paletavimas.DO_New_box -> Conveyor_RND_SC.DI_New_Box
  Paint_Blue.DO_Ready -> Paletavimas.DI_BlueReady
  Paint_Blue.DO_TCP_TRACE -> TraceTCP.Enabled
  Paint_Blue.DO_TCP_CLEAR -> TraceTCP.Clear
  Paint_Red.DO_TCP_TRACE -> TraceTCP_2.Enabled
  Paint_Red.DO_TCP_CLEAR -> TraceTCP_2.Clear
  Paletavimas.DO_Paint_Red_Small -> Paint_Red.DI_Paint_Small
  Paletavimas.DO_Paint_Red_Tall -> Paint_Red.DI_Paint_Tall
  Paletavimas.DO_Paint_Blue_Small -> Paint_Blue.DI_Paint_Small
  Paletavimas.DO_Paint_Blue_Tall -> Paint_Blue.DI_Paint_Tall
  Paletavimas.DO_Enqueue_Small -> Griebtuvas_2.DI_Enque_Small
  Paletavimas.DO_Enqueue_Tall -> Griebtuvas_2.DI_Enque_Tall
  Paletavimas.DO_DeleteALL_Small -> Griebtuvas_2.DI_Delete_Small
  Paletavimas.DO_DeleteALL_Tall -> Griebtuvas_2.DI_Delete_Tall
Targets, tools, work objects and paths stored in the station and not in the controller backup, written as RAPID:
! task T_ROB1
MODULE Module1
  CONST robtarget Didele_ties_piest:=[[-500.000094663,2099.999976261,1150.000241875],[0,-0.706073245,0.708138808,0],[-1,0,0,0],[9E+09,9E+09,9E+09,9E+09,9E+09,9E+09]];
  CONST robtarget Didele_virs_piest:=[[-500.00009482,2100.000045238,1205.091525026],[0,-0.706073245,0.708138808,0],[-1,0,0,0],[9E+09,9E+09,9E+09,9E+09,9E+09,9E+09]];
  CONST robtarget Maza_ties_piest:=[[-1400.000277317,2100.000253447,1100.000411858],[0,-0.706073243,0.708138811,0],[-1,0,0,0],[9E+09,9E+09,9E+09,9E+09,9E+09,9E+09]];
  CONST robtarget Maza_virs_piest:=[[-1400.000277317,2100.00034861,1144.065558591],[0,-0.706073227,0.708138826,0],[-1,0,0,0],[9E+09,9E+09,9E+09,9E+09,9E+09,9E+09]];
  CONST robtarget Didele_ties_conveyor:=[[2504.292,960.385,809],[0,0,1,0],[-2,0,0,0],[9E+09,9E+09,9E+09,9E+09,9E+09,9E+09]];
  CONST robtarget Maza_pries_piesima:=[[-200.095627935,1365.111929006,1486.920311485],[0,-0.706073231,0.708138822,0],[-1,0,0,0],[9E+09,9E+09,9E+09,9E+09,9E+09,9E+09]];
  CONST robtarget Didele_pries_piesima:=[[-876.40010473,1225.00022946,1665.000321221],[0,-0.706073245,0.708138808,0],[-1,0,0,0],[9E+09,9E+09,9E+09,9E+09,9E+09,9E+09]];
  CONST robtarget Maza_ties_conveyor:=[[1443.841,905.155,755.519],[0,0,1,0],[-2,0,0,0],[9E+09,9E+09,9E+09,9E+09,9E+09,9E+09]];
  CONST robtarget Didele_1:=[[2505.32,794.624,809],[0,-0.707106781,0.707106781,0],[-2,0,-1,0],[9E+09,9E+09,9E+09,9E+09,9E+09,9E+09]];
  CONST robtarget Maza_1:=[[1405.32,794.624,759],[0,-0.707106781,0.707106781,0],[0,0,0,0],[9E+09,9E+09,9E+09,9E+09,9E+09,9E+09]];
  PROC Deze_Tall_iki_konvejerio()
    MoveL Home,v1000,z100,tVacuum\WObj:=wobj0;
    MoveL Didele_pries_piesima,v1000,z100,tVacuum\WObj:=wobj0;
    MoveL Didele_ties_piest,v1000,z100,tVacuum\WObj:=wobj0;
    MoveL Didele_virs_piest,v1000,z100,tVacuum\WObj:=wobj0;
    MoveJ Didele_ties_conveyor,v1000,z100,tVacuum\WObj:=wobj0;
  ENDPROC
  PROC Deze_Small_iki_konvejerio()
    MoveL Home,v1000,z100,tVacuum\WObj:=wobj0;
    MoveL Maza_pries_piesima,v1000,z100,tVacuum\WObj:=wobj0;
    MoveL Maza_ties_piest,v1000,z100,tVacuum\WObj:=wobj0;
    MoveL Maza_virs_piest,v1000,z100,tVacuum\WObj:=wobj0;
    MoveL Maza_ties_conveyor,v1000,z100,tVacuum\WObj:=wobj0;
    MoveL Maza_ties_conveyor,v1000,z100,tVacuum\WObj:=wobj0;
  ENDPROC
  PROC Deze_Small_iki_padeklo()
    MoveJ Home,v1000,z100,tVacuum\WObj:=wobj0;
    MoveJ Maza_virs_paimt,v1000,z100,tVacuum\WObj:=wobj0;
    MoveL Maza_ties_paimt,v1000,z100,tVacuum\WObj:=wobj0;
    MoveL Maza_virs_paimt,v1000,z100,tVacuum\WObj:=wobj0;
    MoveL Home,v1000,z100,tVacuum\WObj:=wobj0;
    MoveJ Maza_pries_piesima,v1000,z100,tVacuum\WObj:=wobj0;
    MoveJ Maza_virs_piest,v1000,z100,tVacuum\WObj:=wobj0;
    MoveL Maza_ties_piest,v1000,z100,tVacuum\WObj:=wobj0;
    MoveL Maza_ties_piest,v1000,z100,tVacuum\WObj:=wobj0;
    MoveJ Maza_pries_piesima,v1000,z100,tVacuum\WObj:=wobj0;
    MoveJ Home,v1000,z100,tVacuum\WObj:=wobj0;
  ENDPROC
  PROC Deze_Tall_iki_padeklo()
    MoveL Home,v1000,z100,tVacuum\WObj:=wobj0;
    MoveL Didele_virs_paimt,v1000,z100,tVacuum\WObj:=wobj0;
    MoveL Didele_ties_paimt,v1000,z100,tVacuum\WObj:=wobj0;
    MoveL Didele_virs_paimt,v1000,z100,tVacuum\WObj:=wobj0;
    MoveL Home,v1000,z100,tVacuum\WObj:=wobj0;
    MoveJ Didele_pries_piesima,v1000,z100,tVacuum\WObj:=wobj0;
    MoveL Didele_virs_piest,v1000,z100,tVacuum\WObj:=wobj0;
    MoveL Didele_ties_piest,v1000,z100,tVacuum\WObj:=wobj0;
    MoveL Didele_virs_piest,v1000,z100,tVacuum\WObj:=wobj0;
    MoveJ Didele_pries_piesima,v1000,z100,tVacuum\WObj:=wobj0;
    MoveJ Home,v1000,z100,tVacuum\WObj:=wobj0;
  ENDPROC
  PROC Dezes_Pattern()
    MoveL Didele_1,v1000,z100,tVacuum\WObj:=wobj0;
    MoveL Maza_1,v1000,z100,tVacuum\WObj:=wobj0;
  ENDPROC
  PROC Virs()
    MoveL Virs_Paleciu,v1000,z100,tVacuum\WObj:=wobj0;
  ENDPROC
ENDMODULE


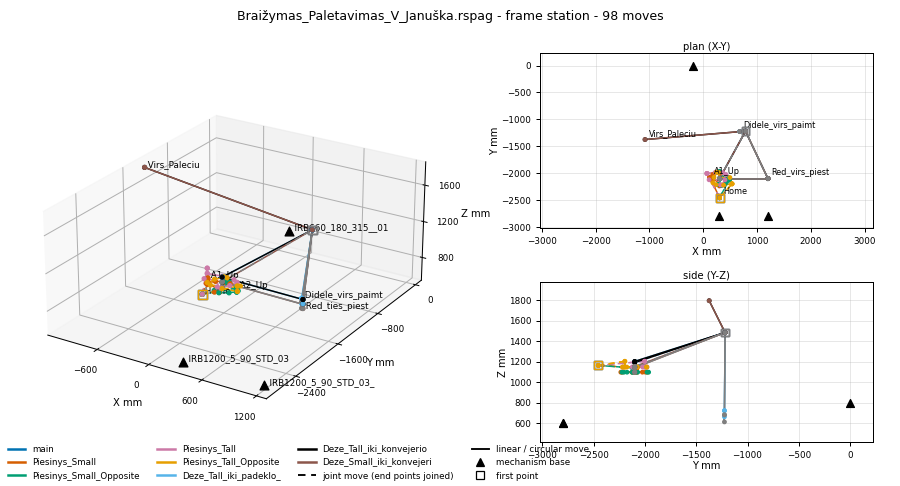
[picture p0: tool path of Braižymas_Paletavimas_V_Januška.rspag in frame station, 98 of 108 moves have a stored position in this frame; points joined in program order, loops and branches not executed]
--- Backups/Paint_Blue/RAPID/TASK1/PROGMOD/CalibData.mod ---
MODULE CalibData
    TASK PERS wobjdata Small_Dezes_Wobj:=[FALSE,TRUE,"",[[700,-800,-200],[0.707107,0,0,0.707107]],[[1050,150,700],[6.12323E-17,0,0,1]]];
    TASK PERS wobjdata Small_Dezes_Wobj_Op:=[FALSE,TRUE,"",[[0.137,-2.682,-3.962],[1,0,0,0]],[[849.863,-247.318,503.962],[0.707106781,0,0,0.707106781]]];
    TASK PERS wobjdata Tall_Dezes_Wobj:=[FALSE,TRUE,"",[[550,250,550],[0.707106781,0,0,-0.707106781]],[[0,0,0],[1,0,0,0]]];
    TASK PERS wobjdata Tall_Dezes_Wobj_Op:=[FALSE,TRUE,"",[[-3.512,-14.105,1.505],[1,0,0,0]],[[853.512,-235.895,548.495],[0.707106781,0,0,0.707106781]]];
    PERS tooldata Pen_TCP:=[TRUE,[[110,0,140],[0.707106781,0,0.707106781,0]],[1,[10.7435139,0,140],[1,0,0,0],0,0,0]];
ENDMODULE

--- Backups/Paint_Blue/RAPID/TASK1/PROGMOD/MainModule.mod ---
MODULE MainModule
    CONST robtarget Home:=[[345.177503635,-2.35947031,565.925003928],[-0.000000009,0.000000008,1,0.000000009],[-1,-1,0,1],[9E+09,9E+09,9E+09,9E+09,9E+09,9E+09]];
    CONST robtarget A1_Up:=[[71.412982699,172.917001677,42.514055788],[0,-0.707106781,0.707106781,0],[0,0,-1,1],[9E+09,9E+09,9E+09,9E+09,9E+09,9E+09]];
    CONST robtarget A1:=[[71.413,172.917,0],[0,-0.707106781,0.707106781,0],[0,0,-1,1],[9E+09,9E+09,9E+09,9E+09,9E+09,9E+09]];
    CONST robtarget A_B1:=[[75,150,0],[0,-0.707106781,0.707106781,0],[0,0,-1,1],[9E+09,9E+09,9E+09,9E+09,9E+09,9E+09]];
    CONST robtarget B1:=[[74.394,140.485,0],[0,-0.707106781,0.707106781,0],[0,0,-1,1],[9E+09,9E+09,9E+09,9E+09,9E+09,9E+09]];
    CONST robtarget C1:=[[97.561,121.951,0],[0,-0.707106781,0.707106781,0],[0,0,-1,1],[9E+09,9E+09,9E+09,9E+09,9E+09,9E+09]];
    CONST robtarget C_D1:=[[197.1225,102.0948,0],[0,-0.707106781,0.707106781,0],[0,0,-1,1],[9E+09,9E+09,9E+09,9E+09,9E+09,9E+09]];
    CONST robtarget D1:=[[248.32,14.395,0],[0,-0.707106781,0.707106781,0],[0,0,-1,1],[9E+09,9E+09,9E+09,9E+09,9E+09,9E+09]];
    CONST robtarget E1:=[[292.04,30.135,0],[0,-0.707106781,0.707106781,0],[-1,-1,0,1],[9E+09,9E+09,9E+09,9E+09,9E+09,9E+09]];
    CONST robtarget E_F1:=[[229.2262,150,0],[0,-0.707106781,0.707106781,0],[0,0,-1,1],[9E+09,9E+09,9E+09,9E+09,9E+09,9E+09]];
    CONST robtarget F1:=[[274.148,255.256,0],[0,-0.707106781,0.707106781,0],[-1,-1,0,1],[9E+09,9E+09,9E+09,9E+09,9E+09,9E+09]];
    CONST robtarget G1:=[[208.333,275,0],[0,-0.707106781,0.707106781,0],[0,0,-1,1],[9E+09,9E+09,9E+09,9E+09,9E+09,9E+09]];
    CONST robtarget H1:=[[125,225,0],[0,-0.707106781,0.707106781,0],[0,0,-1,1],[9E+09,9E+09,9E+09,9E+09,9E+09,9E+09]];
    CONST robtarget H_A1:=[[101.6006,195.4662,0],[0,-0.707106781,0.707106781,0],[0,0,-1,1],[9E+09,9E+09,9E+09,9E+09,9E+09,9E+09]];
    CONST robtarget A2_Up:=[[71.412982699,172.917001677,42.514055788],[0,0.707106781,0.707106781,0],[-1,-1,0,1],[9E+09,9E+09,9E+09,9E+09,9E+09,9E+09]];
    CONST robtarget A2:=[[71.413,172.917,0],[0,0.707106781,0.707106781,0],[-1,-1,0,1],[9E+09,9E+09,9E+09,9E+09,9E+09,9E+09]];
    CONST robtarget A_B2:=[[75,150,0],[0,0.707106781,0.707106781,0],[-1,-1,0,1],[9E+09,9E+09,9E+09,9E+09,9E+09,9E+09]];
    CONST robtarget B2:=[[74.394,140.485,0],[0,0.707106781,0.707106781,0],[-1,-1,0,1],[9E+09,9E+09,9E+09,9E+09,9E+09,9E+09]];
    CONST robtarget C2:=[[97.561,121.951,0],[0,0.707106781,0.707106781,0],[-1,-1,0,1],[9E+09,9E+09,9E+09,9E+09,9E+09,9E+09]];
    CONST robtarget C_D2:=[[197.1225,102.0948,0],[0,0.707106781,0.707106781,0],[-1,-1,0,1],[9E+09,9E+09,9E+09,9E+09,9E+09,9E+09]];
    CONST robtarget D2:=[[248.32,14.395,0],[0,0.707106781,0.707106781,0],[-1,-1,0,1],[9E+09,9E+09,9E+09,9E+09,9E+09,9E+09]];
    CONST robtarget E2:=[[292.04,30.135,0],[0,0.707106781,0.707106781,0],[0,0,-1,1],[9E+09,9E+09,9E+09,9E+09,9E+09,9E+09]];
    CONST robtarget E_F2:=[[229.2262,150,0],[0,0.707106781,0.707106781,0],[-1,-1,0,1],[9E+09,9E+09,9E+09,9E+09,9E+09,9E+09]];
    CONST robtarget F2:=[[274.148,255.256,0],[0,0.707106781,0.707106781,0],[0,0,-1,1],[9E+09,9E+09,9E+09,9E+09,9E+09,9E+09]];
    CONST robtarget G2:=[[208.333,275,0],[0,0.707106781,0.707106781,0],[-1,-1,0,1],[9E+09,9E+09,9E+09,9E+09,9E+09,9E+09]];
    CONST robtarget H2:=[[125,225,0],[0,0.707106781,0.707106781,0],[-1,-1,0,1],[9E+09,9E+09,9E+09,9E+09,9E+09,9E+09]];
    CONST robtarget H_A2:=[[101.6006,195.4662,0],[0,0.707106781,0.707106781,0],[-1,-1,0,1],[9E+09,9E+09,9E+09,9E+09,9E+09,9E+09]];
    CONST robtarget Home_2:=[[250.584789459,-34.674605876,704.871446723],[0.000000449,0.000000007,1,0.000000041],[0,-1,0,0],[9E+09,9E+09,9E+09,9E+09,9E+09,9E+09]];
    CONST robtarget A3_Up:=[[17.857108156,246.428586907,56.367244571],[0,-0.707106781,0.707106781,0],[0,0,-1,1],[9E+09,9E+09,9E+09,9E+09,9E+09,9E+09]];
    CONST robtarget A3:=[[17.8571,246.4286,0],[0,-0.707106781,0.707106781,0],[0,0,-1,1],[9E+09,9E+09,9E+09,9E+09,9E+09,9E+09]];
    CONST robtarget B3:=[[57.0165,128.9505,0],[0,-0.707106781,0.707106781,0],[0,0,-1,1],[9E+09,9E+09,9E+09,9E+09,9E+09,9E+09]];
    CONST robtarget B_C3:=[[184.2408,133.1936,0],[0,-0.707106781,0.707106781,0],[0,0,-1,1],[9E+09,9E+09,9E+09,9E+09,9E+09,9E+09]];
    CONST robtarget C3:=[[266.2915,35.8709,0],[0,-0.707106781,0.707106781,0],[-1,-1,0,1],[9E+09,9E+09,9E+09,9E+09,9E+09,9E+09]];
    CONST robtarget D3:=[[307.345,31.7655,0],[0,-0.707106781,0.707106781,0],[-1,-1,0,1],[9E+09,9E+09,9E+09,9E+09,9E+09,9E+09]];
    CONST robtarget D_E3:=[[319.7224,75,0],[0,-0.707106781,0.707106781,0],[-1,-1,0,1],[9E+09,9E+09,9E+09,9E+09,9E+09,9E+09]];
    CONST robtarget E3:=[[351.7609,127.0833,0],[0,-0.707106781,0.707106781,0],[-1,-1,0,1],[9E+09,9E+09,9E+09,9E+09,9E+09,9E+09]];
    CONST robtarget E_F3:=[[352.8,178.8472,0],[0,-0.707106781,0.707106781,0],[-1,-1,0,1],[9E+09,9E+09,9E+09,9E+09,9E+09,9E+09]];
    CONST robtarget F3:=[[371.3761,227.1744,0],[0,-0.707106781,0.707106781,0],[-1,-1,0,1],[9E+09,9E+09,9E+09,9E+09,9E+09,9E+09]];
    CONST robtarget G3:=[[313.6281,261.8231,0],[0,-0.707106781,0.707106781,0],[-1,-1,0,1],[9E+09,9E+09,9E+09,9E+09,9E+09,9E+09]];
    CONST robtarget G_H3:=[[250,244.4829,0],[0,-0.707106781,0.707106781,0],[-1,-1,0,1],[9E+09,9E+09,9E+09,9E+09,9E+09,9E+09]];
    CONST robtarget H3:=[[174.3437,269.9016,0],[0,-0.707106781,0.707106781,0],[0,0,-1,1],[9E+09,9E+09,9E+09,9E+09,9E+09,9E+09]];
    CONST robtarget Home_3:=[[250.584789459,-34.674605876,704.871446723],[0.000000449,0.000000007,1,0.000000041],[0,-1,0,0],[9E+09,9E+09,9E+09,9E+09,9E+09,9E+09]];
    CONST robtarget A4_Up:=[[17.857108156,246.428586907,56.367244571],[0,0.707106781,0.707106781,0],[-1,-1,0,1],[9E+09,9E+09,9E+09,9E+09,9E+09,9E+09]];
    CONST robtarget A4:=[[17.8571,246.4286,0],[0,0.707106781,0.707106781,0],[-1,-1,0,1],[9E+09,9E+09,9E+09,9E+09,9E+09,9E+09]];
    CONST robtarget B4:=[[57.0165,128.9505,0],[0,0.707106781,0.707106781,0],[-1,-1,0,1],[9E+09,9E+09,9E+09,9E+09,9E+09,9E+09]];
    CONST robtarget B_C4:=[[184.2408,133.1936,0],[0,0.707106781,0.707106781,0],[-1,-1,0,1],[9E+09,9E+09,9E+09,9E+09,9E+09,9E+09]];
    CONST robtarget C4:=[[266.2915,35.8709,0],[0,0.707106781,0.707106781,0],[0,0,-1,1],[9E+09,9E+09,9E+09,9E+09,9E+09,9E+09]];
    CONST robtarget D4:=[[307.345,31.7655,0],[0,0.707106781,0.707106781,0],[0,0,-1,1],[9E+09,9E+09,9E+09,9E+09,9E+09,9E+09]];
    CONST robtarget D_E4:=[[319.7224,75,0],[0,0.707106781,0.707106781,0],[0,0,-1,1],[9E+09,9E+09,9E+09,9E+09,9E+09,9E+09]];
    CONST robtarget E4:=[[351.7609,127.0833,0],[0,0.707106781,0.707106781,0],[0,0,-1,1],[9E+09,9E+09,9E+09,9E+09,9E+09,9E+09]];
    CONST robtarget E_F4:=[[352.8,178.8472,0],[0,0.707106781,0.707106781,0],[0,0,-1,1],[9E+09,9E+09,9E+09,9E+09,9E+09,9E+09]];
    CONST robtarget F4:=[[371.3761,227.1744,0],[0,0.707106781,0.707106781,0],[0,0,-1,1],[9E+09,9E+09,9E+09,9E+09,9E+09,9E+09]];
    CONST robtarget G4:=[[313.6281,261.8231,0],[0,0.707106781,0.707106781,0],[0,0,-1,1],[9E+09,9E+09,9E+09,9E+09,9E+09,9E+09]];
    CONST robtarget G_H4:=[[250,244.4829,0],[0,0.707106781,0.707106781,0],[0,0,-1,1],[9E+09,9E+09,9E+09,9E+09,9E+09,9E+09]];
    CONST robtarget H4:=[[174.3437,269.9016,0],[0,0.707106781,0.707106781,0],[-1,-1,0,1],[9E+09,9E+09,9E+09,9E+09,9E+09,9E+09]];
    !RED - SMALL
    PROC main()
        SetDO DO_RotLeft, 1;
        SetDO DO_RotLeft, 0;
        MoveJ Home,v5000,fine,Pen_TCP\WObj:=wobj0;
        SetDO DO_Ready, 1;
        SetDO DO_BoxDone, 0;
        SetDO DO_AttachBox, 0;
        SetDO DO_TCP_TRACE, 0;
        WHILE TRUE DO
            WaitUntil (DI_Paint_Small = 1 OR DI_Paint_Tall = 1);
            SetDO DO_Ready, 0;
            SetDO DO_AttachBox, 1;
            WaitDI DI_RotationDone, 1;
            IF DI_Paint_Tall = 1 THEN
                Piesinys_Tall;
            ELSEIF DI_Paint_Small = 1 THEN
                Piesinys_Small;
            ENDIF
            WaitRob\inpos;
            SetDO DO_RotRight, 1;
            WaitTime 0.5;
            WaitDI DI_RotationDone, 1;
            SetDO DO_RotRight, 0;
            IF DI_Paint_Tall = 1 THEN
                Piesinys_Tall;
            ELSEIF DI_Paint_Small = 1 THEN
                Piesinys_Small;
            ENDIF
            WaitRob\inpos;
            SetDO DO_RotLeft, 1;
            WaitTime 0.5;
            WaitDI DI_RotationDone, 1;
            SetDO DO_RotLeft, 0;
            SetDO DO_AttachBox, 0;
            SetDO DO_BoxDone, 1;
            WaitTime 0.5;
            WaitDI DI_PositionerFree, 1;
            SetDO DO_Ready, 1;
            SetDO DO_BoxDone, 0;
        ENDWHILE
    ENDPROC
    PROC Piesinys_Small()
        MoveJ Home,v5000,fine,Pen_TCP\WObj:=wobj0;
        MoveJ A1_Up,v1000,fine,Pen_TCP\WObj:=Small_Dezes_Wobj;
        WaitDI DI_RotationDone, 1;
        MoveL A1,v1000,fine,Pen_TCP\WObj:=Small_Dezes_Wobj;
        SetDO DO_TCP_TRACE, 1;
        MoveC A_B1,B1,v1000,fine,Pen_TCP\WObj:=Small_Dezes_Wobj;
        MoveL C1,v1000,fine,Pen_TCP\WObj:=Small_Dezes_Wobj;
        MoveC C_D1,D1,v1000,fine,Pen_TCP\WObj:=Small_Dezes_Wobj;
        MoveL E1,v1000,fine,Pen_TCP\WObj:=Small_Dezes_Wobj;
        MoveC E_F1,F1,v1000,fine,Pen_TCP\WObj:=Small_Dezes_Wobj;
        MoveL G1,v1000,fine,Pen_TCP\WObj:=Small_Dezes_Wobj;
        MoveL H1,v1000,fine,Pen_TCP\WObj:=Small_Dezes_Wobj;
        MoveC H_A1,A1,v1000,fine,Pen_TCP\WObj:=Small_Dezes_Wobj;
        SetDO DO_TCP_TRACE, 0;
        MoveL A1_Up,v1000,fine,Pen_TCP\WObj:=Small_Dezes_Wobj;
        MoveJ Home,v5000,fine,Pen_TCP\WObj:=wobj0;
        PulseDO DO_TCP_CLEAR;
    ENDPROC
    PROC Piesinys_Small_Opposite()
        MoveJ Home,v5000,fine,Pen_TCP\WObj:=wobj0;
        MoveJ A2_Up,v1000,fine,Pen_TCP\WObj:=Small_Dezes_Wobj_Op;
        WaitDI DI_RotationDone, 1;
        MoveL A2,v1000,fine,Pen_TCP\WObj:=Small_Dezes_Wobj_Op;
        SetDO DO_TCP_TRACE, 1;
        MoveC A_B2,B2,v1000,fine,Pen_TCP\WObj:=Small_Dezes_Wobj_Op;
        MoveL C2,v1000,fine,Pen_TCP\WObj:=Small_Dezes_Wobj_Op;
        MoveC C_D2,D2,v1000,fine,Pen_TCP\WObj:=Small_Dezes_Wobj_Op;
        MoveL E2,v1000,fine,Pen_TCP\WObj:=Small_Dezes_Wobj_Op;
        MoveC E_F2,F2,v1000,fine,Pen_TCP\WObj:=Small_Dezes_Wobj_Op;
        MoveL G2,v1000,fine,Pen_TCP\WObj:=Small_Dezes_Wobj_Op;
        MoveL H2,v1000,fine,Pen_TCP\WObj:=Small_Dezes_Wobj_Op;
        MoveC H_A2,A2,v1000,fine,Pen_TCP\WObj:=Small_Dezes_Wobj_Op;
        SetDO DO_TCP_TRACE, 0;
        MoveL A2_Up,v1000,fine,Pen_TCP\WObj:=Small_Dezes_Wobj_Op;
        MoveJ Home,v5000,fine,Pen_TCP\WObj:=wobj0;
        PulseDO DO_TCP_CLEAR;
    ENDPROC
    PROC Piesinys_Tall()
        MoveJ Home,v5000,fine,Pen_TCP\WObj:=wobj0;
        MoveJ A3_Up,v1000,fine,Pen_TCP\WObj:=Tall_Dezes_Wobj;
        WaitDI DI_RotationDone,1;
        MoveL A3,v1000,fine,Pen_TCP\WObj:=Tall_Dezes_Wobj;
        SetDO DO_TCP_TRACE,1;
        MoveL B3,v1000,fine,Pen_TCP\WObj:=Tall_Dezes_Wobj;
        MoveC B_C3,C3,v1000,fine,Pen_TCP\WObj:=Tall_Dezes_Wobj;
        MoveL D3,v1000,fine,Pen_TCP\WObj:=Tall_Dezes_Wobj;
        MoveC D_E3,E3,v1000,fine,Pen_TCP\WObj:=Tall_Dezes_Wobj;
        MoveC E_F3,F3,v1000,fine,Pen_TCP\WObj:=Tall_Dezes_Wobj;
        MoveL G3,v1000,fine,Pen_TCP\WObj:=Tall_Dezes_Wobj;
        MoveC G_H3,H3,v1000,fine,Pen_TCP\WObj:=Tall_Dezes_Wobj;
        MoveL A3,v1000,fine,Pen_TCP\WObj:=Tall_Dezes_Wobj;
        SetDO DO_TCP_TRACE,0;
        MoveL A3_Up,v1000,fine,Pen_TCP\WObj:=Tall_Dezes_Wobj;
        MoveJ Home,v5000,fine,Pen_TCP\WObj:=wobj0;
        PulseDO DO_TCP_CLEAR;
    ENDPROC
    PROC Piesinys_Tall_Opposite()
        MoveJ Home,v5000,fine,Pen_TCP\WObj:=wobj0;
        MoveJ A4_Up,v1000,fine,Pen_TCP\WObj:=Tall_Dezes_Wobj_Op;
        WaitDI DI_RotationDone,1;
        MoveL A4,v1000,fine,Pen_TCP\WObj:=Tall_Dezes_Wobj_Op;
        SetDO DO_TCP_TRACE,1;
        WaitDO DO_TCP_TRACE,1;
        MoveL B4,v1000,fine,Pen_TCP\WObj:=Tall_Dezes_Wobj_Op;
        MoveC B_C4,C4,v1000,fine,Pen_TCP\WObj:=Tall_Dezes_Wobj_Op;
        MoveL D4,v1000,fine,Pen_TCP\WObj:=Tall_Dezes_Wobj_Op;
        MoveC D_E4,E4,v1000,fine,Pen_TCP\WObj:=Tall_Dezes_Wobj_Op;
        MoveC E_F4,F4,v1000,fine,Pen_TCP\WObj:=Tall_Dezes_Wobj_Op;
        MoveL G4,v1000,fine,Pen_TCP\WObj:=Tall_Dezes_Wobj_Op;
        MoveC G_H4,H4,v1000,fine,Pen_TCP\WObj:=Tall_Dezes_Wobj_Op;
        MoveL A4,v1000,fine,Pen_TCP\WObj:=Tall_Dezes_Wobj_Op;
        SetDO DO_TCP_TRACE,0;
        MoveL A4_Up,v1000,fine,Pen_TCP\WObj:=Tall_Dezes_Wobj_Op;
        MoveJ Home,v5000,fine,Pen_TCP\WObj:=wobj0;
        PulseDO DO_TCP_CLEAR;
    ENDPROC
ENDMODULE

--- Backups/Paletavimas/RAPID/TASK1/PROGMOD/CalibData.mod ---
MODULE CalibData
    PERS tooldata tVacuum:=[TRUE,[[0,0,200],[1,0,0,0]],[18,[0,0,133.333333333],[1,0,0,0],0,0,0]];
ENDMODULE

--- Backups/Paletavimas/RAPID/TASK1/PROGMOD/MainModule.mod ---
MODULE MainModule
    CONST robtarget Virs_Paleciu:=[[881.981068513,1373.703898608,1797.389050372],[0,-0.706073234,0.70813882,0],[0,0,-1,0],[9E+09,9E+09,9E+09,9E+09,9E+09,9E+09]];
    CONST robtarget Didele_virs_paimt:=[[-876.400428231,1224.999729409,724.705783202],[0,-0.706073209,0.708138845,0],[-1,0,0,0],[9E+09,9E+09,9E+09,9E+09,9E+09,9E+09]];
    CONST robtarget Didele_ties_paimt:=[[-876.400327564,1224.999728066,665.000029338],[0,-0.706073209,0.708138845,0],[-1,0,0,0],[9E+09,9E+09,9E+09,9E+09,9E+09,9E+09]];
    CONST robtarget Home:=[[-982.878851174,1218.822752071,1486.920305333],[0,-0.706073209,0.708138845,0],[-1,0,0,0],[9E+09,9E+09,9E+09,9E+09,9E+09,9E+09]];
    CONST robtarget Blue_virs_piest:=[[-500.00009482,2100.000045238,1155.091525026],[0,-0.706073245,0.708138808,0],[-1,0,0,0],[9E+09,9E+09,9E+09,9E+09,9E+09,9E+09]];!Bad
    CONST robtarget Blue_ties_piest:=[[-500.000094663,2099.999976261,1100.000241875],[0,-0.706073245,0.708138808,0],[-1,0,0,0],[9E+09,9E+09,9E+09,9E+09,9E+09,9E+09]];!Bad
    CONST robtarget Red_ties_piest:=[[-1400.000277317,2100.000253447,1100.000411858],[0,-0.706073243,0.708138811,0],[-1,0,0,0],[9E+09,9E+09,9E+09,9E+09,9E+09,9E+09]];!Good
    CONST robtarget Red_virs_piest:=[[-1400.000277317,2100.00034861,1144.065558591],[0,-0.706073227,0.708138826,0],[-1,0,0,0],[9E+09,9E+09,9E+09,9E+09,9E+09,9E+09]];!Good
    CONST robtarget Maza_virs_paimt:=[[-876.400083461,1224.999641133,683.835933858],[0,-0.706073212,0.708138842,0],[-1,0,0,0],[9E+09,9E+09,9E+09,9E+09,9E+09,9E+09]];
    CONST robtarget Maza_ties_paimt:=[[-876.400078213,1224.999641049,614.999844809],[0,-0.706073212,0.708138842,0],[-1,0,0,0],[9E+09,9E+09,9E+09,9E+09,9E+09,9E+09]];
    CONST robtarget Didele_ties_palete:=[[2505.32,794.624,809],[0,-0.707106781,0.707106781,0],[-2,0,-1,0],[9E+09,9E+09,9E+09,9E+09,9E+09,9E+09]];
    CONST robtarget Maza_ties_palete:=[[1405.32,794.624,759],[0,-0.707106781,0.707106781,0],[0,0,0,0],[9E+09,9E+09,9E+09,9E+09,9E+09,9E+09]];

    VAR num delta_x1_Small;
    VAR num delta_y1_Small;
    VAR num delta_z1_Small;
    VAR num delta_x1_Tall;
    VAR num delta_y1_Tall;
    VAR num delta_z1_Tall;
    VAR num delta_z2_Tall;! := 20;
    VAR num delta_z3_Tall;! := 200;
    VAR num delta_z2_Small;! := 20;
    VAR num delta_z3_Small;! := 200;
    VAR num Rotz_Small;
    VAR num Rotz_Tall;
    VAR num delta_virs;

    VAR num dezes_aukstis_Small := 200;
    VAR num dezes_aukstis_Tall := 250;

    PROC main()

        VAR bool pirmas_kartas := TRUE;



        VAR num i;
        VAR num sluoksnis_tall := 0;
        VAR num sluoksnis_small := 0;
        VAR num kelintas_tall := 1;
        VAR num kelintas_small := 1;
        VAR num sluoksniu_skaicius_small := 4;
        VAR num sluoksniu_skaicius_tall := 4;
        VAR bool notDone := TRUE;
        VAR num delta_x1_Small;
        VAR num delta_y1_Small;
        VAR num delta_z1_Small := 0;
        VAR num dezes_aukstis_Small := 200;
        VAR num dezes_aukstis_Tall := 250;

        VAR num Rotz;

        VAR num Kiek_paleciu_kraut:= 4;
        VAR num Sukrauta:= 0;


        VAR bool RedSmall := FALSE;
        VAR bool BlueSmall := FALSE;
        VAR bool RedTall := FALSE;
        VAR bool BlueTall := FALSE;
        SetDO DO_Paint_Blue_Small, 0;
        WaitDO DO_Paint_Blue_Small, 0;
        SetDO DO_Paint_Blue_Tall, 0;
        WaitDO DO_Paint_Blue_Tall, 0;
        SetDO DO_Paint_Red_Small, 0;
        WaitDO DO_Paint_Red_Small, 0;
        SetDO DO_Paint_Red_Tall, 0;
        WaitDO DO_Paint_Red_Tall, 0;
        SetDO DO_Add, 0;

        WHILE Sukrauta < Kiek_paleciu_kraut DO
            WaitUntil((DI_Box_InPlace_Small=1 OR DI_Box_InPlace_Tall=1) AND (DI_RedReady=1 OR DI_BlueReady = 1)) OR
            (DI_BlueDone=1 OR DI_RedDone=1);
            WaitTime 0.001; !Wait if Small Box False pulse has been received
            IF (DI_Box_InPlace_Small=1 AND DI_RedReady=1 AND RedSmall = FALSE AND RedTall = FALSE) THEN
                Deze_Small_iki_padeklo_ 1;
                RedSmall := TRUE;
            ELSEIF (DI_Box_InPlace_Small=1 AND DI_BlueReady=1 AND BlueSmall = FALSE AND BlueTall = FALSE) THEN
                Deze_Small_iki_padeklo_ 2;
                BlueSmall := TRUE;
            ELSEIF (DI_Box_InPlace_Tall=1 AND DI_BlueReady=1 AND BlueSmall = FALSE AND BlueTall = FALSE) THEN
                Deze_Tall_iki_padeklo_ 1;
                BlueTall := TRUE;
            ELSEIF (DI_Box_InPlace_Tall=1 AND DI_RedReady=1 AND RedSmall = FALSE AND RedTall = FALSE) THEN
                Deze_Tall_iki_padeklo_ 2;
                RedTall := TRUE;
            ENDIF
            IF (DI_BlueDone=1 AND DO_Paint_Blue_Tall=1) OR (DI_RedDone=1 AND DO_Paint_Red_Tall=1) THEN
                RedTall := FALSE;
                BlueTall := FALSE;
                Deze_Tall_iki_konvejerio_ sluoksnis_tall, kelintas_tall;
                !Sluoksnio_krovimas_Tall sluoksnis_tall, kelintas_tall;
                IF sluoksnis_tall = (sluoksniu_skaicius_tall-1) AND kelintas_tall = 6 THEN
                    SetDO DO_DeleteALL_tall, 1;
                    sluoksnis_tall := 0;
                    kelintas_tall := 1;
                    SetDO DO_DeleteALL_tall, 0;
                    Sukrauta := Sukrauta + 1;
                ELSEIF kelintas_tall = 6 THEN
                    kelintas_tall := 1;
                    sluoksnis_tall := sluoksnis_tall + 1;
                ELSE
                    kelintas_tall := kelintas_tall + 1;
                ENDIF
            ELSEIF (DI_BlueDone=1 AND DO_Paint_Blue_Small=1) OR (DI_RedDone=1 AND DO_Paint_Red_Small=1) THEN
                RedSmall := FALSE;
                BlueSmall := FALSE;
                Deze_Small_iki_konvejerio_ sluoksnis_small, kelintas_small;
                !Sluoksnio_krovimas_Small sluoksnis_small, kelintas_small;
                IF sluoksnis_small = (sluoksniu_skaicius_small-1) AND kelintas_small = 6 THEN
                    SetDO DO_DeleteALL_Small, 1;
                    sluoksnis_small := 0;
                    kelintas_small := 1;
                    SetDO DO_DeleteALL_Small, 0;
                    Sukrauta := Sukrauta + 1;
                ELSEIF kelintas_small = 6 THEN
                    kelintas_small := 1;
                    sluoksnis_small := sluoksnis_small + 1;
                ELSE
                    kelintas_small := kelintas_small + 1;
                ENDIF
            ENDIF
        ENDWHILE
        SetDO DO_Paint_Blue_Small, 0;
        WaitDO DO_Paint_Blue_Small, 0;
        SetDO DO_Paint_Blue_Tall, 0;
        WaitDO DO_Paint_Blue_Tall, 0;
        SetDO DO_Paint_Red_Small, 0;
        WaitDO DO_Paint_Red_Small, 0;
        SetDO DO_Paint_Red_Tall, 0;
        WaitDO DO_Paint_Red_Tall, 0;
        SetDO DO_Add, 0;
        Sukrauta := 0;
        MoveL Home,v1000,fine,tVacuum\WObj:=wobj0;

    ENDPROC

    PROC Deze_Tall_iki_padeklo_(num Padeklas)
        SetDO DO_Add, 0;
        MoveJ Home,v7000,z100,tVacuum\WObj:=wobj0;
        MoveL Didele_virs_paimt,v7000,fine,tVacuum\WObj:=wobj0;
        MoveL Didele_ties_paimt,v1000,fine,tVacuum\WObj:=wobj0;
        WaitRob\InPos;
        SetDO DO_Add, 1;
        MoveL Didele_virs_paimt,v3000,fine,tVacuum\WObj:=wobj0;
        MoveL Home,v1000,fine,tVacuum\WObj:=wobj0;
        TEST Padeklas
            CASE 1:
                !Blue padeklas
                MoveL Offs(Blue_virs_piest, 0, 0, 50),v7000,fine,tVacuum\WObj:=wobj0;
                MoveL Offs(Blue_ties_piest, 0, 0, 50),v1000,fine,tVacuum\WObj:=wobj0;
                SetDO DO_Add, 0;
                MoveL Offs(Blue_virs_piest, 0, 0, 50),v3000,fine,tVacuum\WObj:=wobj0;
                SetDO DO_Paint_Blue_Tall, 1;
            CASE 2:
                !Red padeklas
                MoveL Offs(Red_virs_piest,0,0,50),v7000,fine,tVacuum\WObj:=wobj0;
                MoveL Offs(Red_ties_piest,0,0,50),v1000,fine,tVacuum\WObj:=wobj0;
                SetDO DO_Add, 0;
                MoveL Offs(Red_virs_piest,0,0,50),v3000,fine,tVacuum\WObj:=wobj0;
                SetDO DO_Paint_Red_Tall, 1;
        ENDTEST
        MoveJ Home,v7000,z100,tVacuum\WObj:=wobj0;
        WaitRob\InPos;
    ENDPROC
    PROC Deze_Tall_iki_konvejerio_(num sluoksnis_tall, num kelintas_tall)
        delta_z3_Tall := dezes_aukstis_Tall*sluoksnis_tall;
        delta_z2_Tall := delta_z3_Tall + 20;
        delta_z1_Tall := delta_z3_Tall + 500;
        delta_virs := 1000;
        MoveL Home,v7000,z100,tVacuum\WObj:=wobj0;
        IF DI_RedDone = 1 THEN
            SetDO DO_Paint_Red_Tall, 0;
            MoveL Offs(Red_virs_piest, 0, 0, 50),v7000,fine,tVacuum\WObj:=wobj0;
            MoveL Offs(Red_ties_piest, 0, 0, 50),v1000,fine,tVacuum\WObj:=wobj0;
            WaitRob\InPos;
            SetDO DO_Add, 1;
            MoveL Offs(Red_virs_piest, 0, 0, 50),v3000,fine,tVacuum\WObj:=wobj0;
        ELSEIF DI_BlueDone = 1 THEN
            SetDO DO_Paint_Blue_Tall, 0;
            MoveL Offs(Blue_virs_piest, 0, 0, 50),v7000,fine,tVacuum\WObj:=wobj0;
            MoveL Offs(Blue_ties_piest, 0, 0, 50),v1000,fine,tVacuum\WObj:=wobj0;
            WaitRob\InPos;
            SetDO DO_Add, 1;
            MoveL Offs(Blue_virs_piest, 0, 0, 50),v3000,fine,tVacuum\WObj:=wobj0;
        ENDIF
        MoveL Home,v7000,z200,tVacuum\WObj:=wobj0;
        IF sluoksnis_tall MOD 2 = 0 THEN
            TEST kelintas_tall
                CASE 1:
                    delta_x1_Tall := 0;
                    delta_y1_Tall := 0;
                    Rotz_Tall := 0;
                CASE 2:
                    delta_x1_Tall := -300;
                CASE 3:
                    delta_x1_Tall := -600;
                CASE 4:
                    delta_x1_Tall := -900;
                CASE 5:
                    Rotz_Tall := 90;
                    delta_y1_Tall := 400;
                    delta_x1_Tall := -150;
                CASE 6:
                    delta_x1_Tall := -750;
            ENDTEST
        ELSE
            TEST kelintas_tall
                CASE 1:
                    delta_y1_Tall := -100;
                    delta_x1_Tall := -150;
                CASE 2:
                    delta_x1_Tall := -750;
                CASE 3:
                    Rotz_Tall := 0;
                    delta_y1_Tall := 300;
                    delta_x1_Tall := 0;
                CASE 4:
                    delta_x1_Tall := -300;
                CASE 5:
                    delta_x1_Tall := -600;
                CASE 6:
                    delta_x1_Tall := -900;
            ENDTEST
        ENDIF
        MoveL Virs_Paleciu,v7000,z200,tVacuum\WObj:=wobj0;
        WaitDI DI_Pallet_InPlace_Tall, 1;
        PulseDO DO_Enqueue_Tall;
        MoveL RelTool(Didele_ties_palete, delta_x1_Tall, delta_y1_Tall, -delta_virs \Rz:= Rotz_Tall),v7000,fine,tVacuum\WObj:=wobj0;
        MoveL RelTool(Didele_ties_palete, delta_x1_Tall, delta_y1_Tall, -delta_z2_tall \Rz:= Rotz_Tall),v3000,fine,tVacuum\WObj:=wobj0;
        MoveL RelTool(Didele_ties_palete, delta_x1_Tall, delta_y1_Tall, -delta_z3_tall \Rz:= Rotz_Tall),v1000,fine,tVacuum\WObj:=wobj0;
        WaitRob\InPos;
        SetDO DO_Add, 0;
        MoveL RelTool(Didele_ties_palete, delta_x1_Tall, delta_y1_Tall, -delta_z2_tall \Rz:= Rotz_Tall),v3000,fine,tVacuum\WObj:=wobj0;
        MoveL RelTool(Didele_ties_palete, delta_x1_Tall, delta_y1_Tall, -delta_virs \Rz:= Rotz_Tall),v7000,fine,tVacuum\WObj:=wobj0;
        MoveL Home,v7000,z200,tVacuum\WObj:=wobj0;
    ENDPROC
    PROC Deze_Small_iki_konvejerio_(num sluoksnis_small, num kelintas_small)
        delta_z3_Small := dezes_aukstis_Small*sluoksnis_small;
        delta_z2_Small := delta_z3_Small + 20;
        delta_z1_Small := delta_z3_Small + 500;
        delta_virs := 1000;
        MoveL Home,v7000,z200,tVacuum\WObj:=wobj0;
        IF DI_RedDone = 1 THEN
            SetDO DO_Paint_Red_Small, 0;
            MoveL Red_virs_piest,v7000,fine,tVacuum\WObj:=wobj0;
            MoveL Red_ties_piest,v1000,fine,tVacuum\WObj:=wobj0;
            WaitRob\InPos;
            SetDO DO_Add, 1;
            MoveL Red_virs_piest,v3000,fine,tVacuum\WObj:=wobj0;
        ELSEIF DI_BlueDone = 1 THEN
            SetDO DO_Paint_Blue_Small, 0;
            MoveL Blue_virs_piest,v7000,fine,tVacuum\WObj:=wobj0;
            MoveL Blue_ties_piest,v1000,fine,tVacuum\WObj:=wobj0;
            WaitRob\InPos;
            SetDO DO_Add, 1;
            MoveL Blue_virs_piest,v3000,fine,tVacuum\WObj:=wobj0;
        ENDIF
        MoveL Home,v7000,z200,tVacuum\WObj:=wobj0;
        IF sluoksnis_Small MOD 2 = 0 THEN
            TEST kelintas_Small
                CASE 1:
                    delta_x1_Small := 0;
                    delta_y1_Small := 0;
                    Rotz_Small := 0;
                CASE 2:
                    delta_x1_Small := -300;
                CASE 3:
                    delta_x1_Small := -600;
                CASE 4:
                    delta_x1_Small := -900;
                CASE 5:
                    Rotz_Small := 90;
                    delta_y1_Small := 400;
                    delta_x1_Small := -150;
                CASE 6:
                    delta_x1_Small := -750;
            ENDTEST
        ELSE
            TEST kelintas_small
                CASE 1:
                    Rotz_Small := 90;
                    delta_y1_Small := -100;
                    delta_x1_Small := -150;
                CASE 2:
                    delta_x1_Small := -750;
                CASE 3:
                    Rotz_Small := 0;
                    delta_y1_Small := 300;
                    delta_x1_Small := 0;
                CASE 4:
                    delta_x1_Small := -300;
                CASE 5:
                    delta_x1_Small := -600;
                CASE 6:
                    delta_x1_Small := -900;
            ENDTEST
        ENDIF
        MoveL Virs_Paleciu,v7000,z200,tVacuum\WObj:=wobj0;
        WaitDI DI_Pallet_InPlace_Small, 1;
        PulseDO DO_Enqueue_Small;
        MoveL RelTool(Maza_ties_palete, delta_x1_Small, delta_y1_Small, -delta_virs \Rz:= Rotz_Small),v7000,fine,tVacuum\WObj:=wobj0;
        MoveL RelTool(Maza_ties_palete, delta_x1_Small, delta_y1_Small, -delta_z2_Small \Rz:= Rotz_Small),v3000,fine,tVacuum\WObj:=wobj0;
        MoveL RelTool(Maza_ties_palete, delta_x1_Small, delta_y1_Small, -delta_z3_Small \Rz:= Rotz_Small),v1000,fine,tVacuum\WObj:=wobj0;
        WaitRob\InPos;
        SetDO DO_Add, 0;
        MoveL RelTool(Maza_ties_palete, delta_x1_Small, delta_y1_Small, -delta_z2_Small \Rz:= Rotz_Small),v3000,fine,tVacuum\WObj:=wobj0;
        MoveL RelTool(Maza_ties_palete, delta_x1_Small, delta_y1_Small, -delta_virs \Rz:= Rotz_Small),v7000,fine,tVacuum\WObj:=wobj0;
        MoveL Home,v7000,z200,tVacuum\WObj:=wobj0;
    ENDPROC
    PROC Deze_Small_iki_padeklo_(num Padeklas)
        SetDO DO_Add, 0;
        MoveJ Home,v7000,z100,tVacuum\WObj:=wobj0;
        MoveL Maza_virs_paimt,v7000,fine,tVacuum\WObj:=wobj0;
        MoveL Maza_ties_paimt,v1000,fine,tVacuum\WObj:=wobj0;
        WaitRob\InPos;
        SetDO DO_Add, 1;
        MoveL Maza_virs_paimt,v3000,fine,tVacuum\WObj:=wobj0;
        MoveL Home,v7000,z100,tVacuum\WObj:=wobj0;
        TEST Padeklas
            CASE 1:
                !Red Padeklas
                MoveL Red_virs_piest,v7000,fine,tVacuum\WObj:=wobj0;
                MoveL Red_ties_piest,v1000,fine,tVacuum\WObj:=wobj0;
                SetDO DO_Add, 0;
                MoveL Red_virs_piest,v3000,fine,tVacuum\WObj:=wobj0;
                SetDO DO_Paint_Red_Small, 1;
            CASE 2:
                !Blue Padeklas
                MoveL Blue_virs_piest,v7000,fine,tVacuum\WObj:=wobj0;
                MoveL Blue_ties_piest,v1000,fine,tVacuum\WObj:=wobj0;
                SetDO DO_Add, 0;
                MoveL Blue_virs_piest,v3000,fine,tVacuum\WObj:=wobj0;
                SetDO DO_Paint_Blue_Small, 1;
        ENDTEST
        MoveJ Home,v7000,z100,tVacuum\WObj:=wobj0;
    ENDPROC
ENDMODULE

--- Backups/Paint_Blue/SYSPAR/EIO.cfg ---
EIO:CFG_1.0:6:1::
#
INDUSTRIAL_NETWORK:

      -Name "DeviceNet" -Label "DeviceNet Master/Slave Network" -Address "2"
#
DEVICENET_INTERNAL_DEVICE:

      -Name "DN_Internal_Device" -VendorName "ABB Robotics"\
      -ProductName "DeviceNet Internal Slave Device"
#
EIO_SIGNAL:

      -Name "DI_Paint_Tall" -SignalType "DI" -DeviceMap "100"

      -Name "DI_PositionerFree" -SignalType "DI" -DeviceMap "101"

      -Name "DI_RotationDone" -SignalType "DI" -DeviceMap "102"

      -Name "DO_AttachBox" -SignalType "DO" -DeviceMap "103"

      -Name "DO_BoxDone" -SignalType "DO" -DeviceMap "104"

      -Name "DO_Ready" -SignalType "DO" -DeviceMap "105"

      -Name "DO_RotHome" -SignalType "DO" -DeviceMap "106"

      -Name "DO_RotLeft" -SignalType "DO" -DeviceMap "107"

      -Name "DO_RotRight" -SignalType "DO" -DeviceMap "108"

      -Name "DO_TCP_TRACE" -SignalType "DO" -DeviceMap "109"

      -Name "DO_TCP_CLEAR" -SignalType "DO" -DeviceMap "110"

      -Name "DI_Paint_Small" -SignalType "DI" -DeviceMap "111"

--- Backups/Paint_Red/SYSPAR/EIO.cfg ---
EIO:CFG_1.0:6:1::
#
INDUSTRIAL_NETWORK:

      -Name "DeviceNet" -Label "DeviceNet Master/Slave Network" -Address "2"
#
DEVICENET_INTERNAL_DEVICE:

      -Name "DN_Internal_Device" -VendorName "ABB Robotics"\
      -ProductName "DeviceNet Internal Slave Device"
#
EIO_SIGNAL:

      -Name "DI_Paint_Small" -SignalType "DI" -DeviceMap "100"

      -Name "DI_PositionerFree" -SignalType "DI" -DeviceMap "101"

      -Name "DI_RotationDone" -SignalType "DI" -DeviceMap "102"

      -Name "DO_AttachBox" -SignalType "DO" -DeviceMap "103"

      -Name "DO_BoxDone" -SignalType "DO" -DeviceMap "104"

      -Name "DO_Ready" -SignalType "DO" -DeviceMap "105"

      -Name "DO_RotHome" -SignalType "DO" -DeviceMap "106"

      -Name "DO_RotLeft" -SignalType "DO" -DeviceMap "107"

      -Name "DO_RotRight" -SignalType "DO" -DeviceMap "108"

      -Name "DO_TCP_TRACE" -SignalType "DO" -DeviceMap "109"

      -Name "DO_TCP_CLEAR" -SignalType "DO" -DeviceMap "110"

      -Name "DI_Paint_Tall" -SignalType "DI" -DeviceMap "111"

--- Backups/Paletavimas/SYSPAR/EIO.cfg ---
EIO:CFG_1.0:6:1::
#
INDUSTRIAL_NETWORK:

      -Name "DeviceNet" -Label "DeviceNet Master/Slave Network" -Address "2"
#
DEVICENET_INTERNAL_DEVICE:

      -Name "DN_Internal_Device" -VendorName "ABB Robotics"\
      -ProductName "DeviceNet Internal Slave Device"
#
EIO_SIGNAL:

      -Name "DI_New_box" -SignalType "DI" -DeviceMap "134"

      -Name "DO_New_box" -SignalType "DO" -DeviceMap "0"

      -Name "DO_New_pallet_Small" -SignalType "DO" -DeviceMap "1"

      -Name "DI_Box_InPlace_Small" -SignalType "DI" -DeviceMap "10"

      -Name "DI_Pallet_InPlace_Small" -SignalType "DI" -DeviceMap "11"

      -Name "DI_Gripper_Opened" -SignalType "DI" -DeviceMap "12"

      -Name "DI_Gripper_closed" -SignalType "DI" -DeviceMap "13"

      -Name "DO_DeleteALL_Tall" -SignalType "DO" -DeviceMap "14"

      -Name "DO_DeleteALL_Small" -SignalType "DO" -DeviceMap "141"

      -Name "DO_New_pallet_Tall" -SignalType "DO" -DeviceMap "142"

      -Name "DI_Box_InPlace_Tall" -SignalType "DI" -DeviceMap "100"

      -Name "DO_Add" -SignalType "DO" -DeviceMap "102"

      -Name "DI_Pallet_InPlace_Tall" -SignalType "DI" -DeviceMap "111"

      -Name "DI_BlueReady" -SignalType "DI" -DeviceMap "133"

      -Name "DI_RedReady" -SignalType "DI" -DeviceMap "135"

      -Name "DI_RedDone" -SignalType "DI" -DeviceMap "155"

      -Name "DI_BlueDone" -SignalType "DI" -DeviceMap "156"

      -Name "DO_Paint_Red_Small" -SignalType "DO" -DeviceMap "157"

      -Name "DO_Paint_Blue_Tall" -SignalType "DO" -DeviceMap "158"

      -Name "DO_Paint_Blue_Small" -SignalType "DO" -DeviceMap "110"

      -Name "DO_Paint_Red_Tall" -SignalType "DO" -DeviceMap "133"

      -Name "DO_Enqueue_Small" -SignalType "DO"

      -Name "DO_Enqueue_Tall" -SignalType "DO"
